LIN {X 0,Y 591.469,Z 583.737,A -85,B 0,C 180,E1 -8891.352,E2 -8891.352} C_VEL
LIN {X 0,Y 591.483,Z 583.74,A -85,B 0,C 180,E1 -8894.195,E2 -8894.195} C_VEL
LIN {X 0,Y 591.491,Z 583.733,A -85,B 0,C 180,E1 -8896.997,E2 -8896.997} C_VEL
LIN {X 0,Y 591.518,Z 583.737,A -85,B 0,C 180,E1 -8899.769,E2 -8899.769} C_VEL
LIN {X 0,Y 591.543,Z 583.729,A -85,B 0,C 180,E1 -8902.516,E2 -8902.516} C_VEL
LIN {X 0,Y 591.625,Z 583.717,A -85,B 0,C 180,E1 -8905.246,E2 -8905.246} C_VEL
LIN {X 0,Y 591.718,Z 583.706,A -85,B 0,C 180,E1 -8909.322,E2 -8909.322} C_VEL
LIN {X 0,Y 591.68,Z 583.711,A -85,B 0,C 180,E1 -8911.357,E2 -8911.357} C_VEL
LIN {X 0,Y 591.625,Z 583.717,A -85,B 0,C 180,E1 -8914.754,E2 -8914.754} C_VEL
LIN {X 0,Y 591.543,Z 583.729,A -85,B 0,C 180,E1 -8917.484,E2 -8917.484} C_VEL
LIN {X 0,Y 591.53,Z 583.729,A -85,B 0,C 180,E1 -8920.638,E2 -8920.638} C_VEL
LIN {X 0,Y 591.518,Z 583.738,A -85,B 0,C 180,E1 -8923.834,E2 -8923.834} C_VEL
LIN {X 0,Y 591.492,Z 583.735,A -85,B 0,C 180,E1 -8926.511,E2 -8926.511} C_VEL
LIN {X 0,Y 591.458,Z 583.739,A -85,B 0,C 180,E1 -8929.365,E2 -8929.365} C_VEL
LIN {X 0,Y 591.478,Z 583.738,A -85,B 0,C 180,E1 -8931.537,E2 -8931.537} C_VEL
LIN {X 0,Y 591.433,Z 583.743,A -85,B 0,C 180,E1 -8934.488,E2 -8934.488} C_VEL
LIN {X 0,Y 591.429,Z 583.744,A -85,B 0,C 180,E1 -8937.509,E2 -8937.509} C_VEL
LIN {X 0,Y 591.468,Z 583.742,A -85,B 0,C 180,E1 -8940.175,E2 -8940.175} C_VEL
LIN {X 0,Y 591.437,Z 583.74,A -85,B 0,C 180,E1 -8943.01,E2 -8943.01} C_VEL
LIN {X 0,Y 591.485,Z 583.737,A -85,B 0,C 180,E1 -8945.469,E2 -8945.469} C_VEL
LIN {X 0,Y 591.444,Z 583.749,A -85,B 0,C 180,E1 -8948.012,E2 -8948.012} C_VEL
LIN {X 0,Y 591.448,Z 583.739,A -85,B 0,C 180,E1 -8950.717,E2 -8950.717} C_VEL
LIN {X 0,Y 591.417,Z 583.744,A -85,B 0,C 180,E1 -8953.387,E2 -8953.387} C_VEL
LIN {X 0,Y 591.427,Z 583.746,A -85,B 0,C 180,E1 -8956.256,E2 -8956.256} C_VEL
LIN {X 0,Y 591.433,Z 583.743,A -85,B 0,C 180,E1 -8958.455,E2 -8958.455} C_VEL
LIN {X 0,Y 591.427,Z 583.743,A -85,B 0,C 180,E1 -8961.412,E2 -8961.412} C_VEL
LIN {X 0,Y 591.476,Z 583.741,A -85,B 0,C 180,E1 -8963.693,E2 -8963.693} C_VEL
LIN {X 0,Y 591.442,Z 583.746,A -85,B 0,C 180,E1 -8966.178,E2 -8966.178} C_VEL
LIN {X 0,Y 591.449,Z 583.74,A -85,B 0,C 180,E1 -8968.595,E2 -8968.595} C_VEL
LIN {X 0,Y 591.486,Z 583.734,A -85,B 0,C 180,E1 -8971.201,E2 -8971.201} C_VEL
LIN {X 0,Y 591.406,Z 583.75,A -85,B 0,C 180,E1 -8974.174,E2 -8974.174} C_VEL
LIN {X 0,Y 591.446,Z 583.744,A -85,B 0,C 180,E1 -8976.256,E2 -8976.256} C_VEL
LIN {X 0,Y 591.471,Z 583.738,A -85,B 0,C 180,E1 -8978.463,E2 -8978.463} C_VEL
LIN {X 0,Y 591.445,Z 583.741,A -85,B 0,C 180,E1 -8981.352,E2 -8981.352} C_VEL
LIN {X 0,Y 591.468,Z 583.742,A -85,B 0,C 180,E1 -8984.195,E2 -8984.195} C_VEL
LIN {X 0,Y 591.506,Z 583.736,A -85,B 0,C 180,E1 -8986.301,E2 -8986.301} C_VEL
LIN {X 0,Y 591.537,Z 583.729,A -85,B 0,C 180,E1 -8989.361,E2 -8989.361} C_VEL
LIN {X 0,Y 591.547,Z 583.728,A -85,B 0,C 180,E1 -8992.516,E2 -8992.516} C_VEL
LIN {X 0,Y 591.544,Z 583.728,A -85,B 0,C 180,E1 -8994.565,E2 -8994.565} C_VEL
LIN {X 0,Y 591.613,Z 583.728,A -85,B 0,C 180,E1 -8995.927,E2 -8995.927} C_VEL
LIN {X 0,Y 591.704,Z 583.708,A -85,B 0,C 180,E1 -8999.322,E2 -8999.322} C_VEL
LIN {X 0,Y 591.669,Z 583.713,A -85,B 0,C 180,E1 -9001.357,E2 -9001.357} C_VEL
LIN {X 0,Y 591.611,Z 583.718,A -85,B 0,C 180,E1 -9004.754,E2 -9004.754} C_VEL
LIN {X 0,Y 591.567,Z 583.724,A -85,B 0,C 180,E1 -9006.8,E2 -9006.8} C_VEL
LIN {X 0,Y 591.504,Z 583.735,A -85,B 0,C 180,E1 -9009.543,E2 -9009.543} C_VEL
LIN {X 0,Y 591.462,Z 583.741,A -85,B 0,C 180,E1 -9011.615,E2 -9011.615} C_VEL
LIN {X 0,Y 591.463,Z 583.74,A -85,B 0,C 180,E1 -9014.4,E2 -9014.4} C_VEL
LIN {X 0,Y 591.43,Z 583.741,A -85,B 0,C 180,E1 -9017.222,E2 -9017.222} C_VEL
LIN {X 0,Y 591.415,Z 583.744,A -85,B 0,C 180,E1 -9019.367,E2 -9019.367} C_VEL
LIN {X 0,Y 591.468,Z 583.741,A -85,B 0,C 180,E1 -9022.269,E2 -9022.269} C_VEL
LIN {X 0,Y 591.407,Z 583.745,A -85,B 0,C 180,E1 -9025.238,E2 -9025.238} C_VEL
LIN {X 0,Y 591.43,Z 583.744,A -85,B 0,C 180,E1 -9027.509,E2 -9027.509} C_VEL
LIN {X 0,Y 591.408,Z 583.752,A -85,B 0,C 180,E1 -9029.83,E2 -9029.83} C_VEL
LIN {X 0,Y 591.407,Z 583.749,A -85,B 0,C 180,E1 -9032.206,E2 -9032.206} C_VEL
LIN {X 0,Y 591.397,Z 583.746,A -85,B 0,C 180,E1 -9034.646,E2 -9034.646} C_VEL
LIN {X 0,Y 591.405,Z 583.744,A -85,B 0,C 180,E1 -9037.159,E2 -9037.159} C_VEL
LIN {X 0,Y 591.404,Z 583.751,A -85,B 0,C 180,E1 -9039.759,E2 -9039.759} C_VEL
LIN {X 0,Y 591.416,Z 583.743,A -85,B 0,C 180,E1 -9042.752,E2 -9042.752} C_VEL
LIN {X 0,Y 591.427,Z 583.747,A -85,B 0,C 180,E1 -9045.673,E2 -9045.673} C_VEL
LIN {X 0,Y 591.392,Z 583.748,A -85,B 0,C 180,E1 -9048.451,E2 -9048.451} C_VEL
LIN {X 0,Y 591.405,Z 583.744,A -85,B 0,C 180,E1 -9051.118,E2 -9051.118} C_VEL
LIN {X 0,Y 591.446,Z 583.745,A -85,B 0,C 180,E1 -9053.691,E2 -9053.691} C_VEL
LIN {X 0,Y 591.423,Z 583.748,A -85,B 0,C 180,E1 -9056.176,E2 -9056.176} C_VEL
LIN {X 0,Y 591.418,Z 583.743,A -85,B 0,C 180,E1 -9058.593,E2 -9058.593} C_VEL
LIN {X 0,Y 591.436,Z 583.741,A -85,B 0,C 180,E1 -9061.21,E2 -9061.21} C_VEL
LIN {X 0,Y 591.401,Z 583.755,A -85,B 0,C 180,E1 -9064.01,E2 -9064.01} C_VEL
LIN {X 0,Y 591.454,Z 583.794,A -85,B 0,C 180,E1 -9066.765,E2 -9066.765} C_VEL
LIN {X 0,Y 593.313,Z 594.595,A -85,B 0,C 180,E1 -9068.533,E2 -9068.533} C_VEL
LIN {X 0,Y 592.679,Z 611.185,A -85,B 0,C 180,E1 -9071.09,E2 -9071.09} C_VEL
LIN {X 0,Y 591.965,Z 630.482,A -85,B 0,C 180,E1 -9074.032,E2 -9074.032} C_VEL
LIN {X 0,Y 591.494,Z 647.827,A -85,B 0,C 180,E1 -9076.649,E2 -9076.649} C_VEL
LIN {X 0,Y 593.595,Z 665.618,A -85,B 0,C 180,E1 -9076.936,E2 -9076.936} C_VEL
LIN {X 0,Y 592.889,Z 754.339,A -85,B 0,C 180,E1 -9078.112,E2 -9078.112} C_VEL
LIN {X 0,Y 592.757,Z 763.761,A -85,B 0,C 180,E1 -9078.303,E2 -9078.303} C_VEL
LIN {X 0,Y 592.554,Z 773.554,A -85,B 0,C 180,E1 -9078.58,E2 -9078.58} C_VEL
LIN {X 0,Y 592.29,Z 784.736,A -85,B 0,C 180,E1 -9079.007,E2 -9079.007} C_VEL
LIN {X 0,Y 592.068,Z 795.202,A -85,B 0,C 180,E1 -9079.52,E2 -9079.52} C_VEL
LIN {X 0,Y 591.759,Z 803.814,A -85,B 0,C 180,E1 -9080.031,E2 -9080.031} C_VEL
LIN {X 0,Y 591.445,Z 813.28,A -85,B 0,C 180,E1 -9080.714,E2 -9080.714} C_VEL
LIN {X 0,Y 591.111,Z 822.077,A -85,B 0,C 180,E1 -9081.482,E2 -9081.482} C_VEL
LIN {X 0,Y 590.911,Z 828.739,A -85,B 0,C 180,E1 -9082.165,E2 -9082.165} C_VEL
LIN {X 0,Y 590.718,Z 835.721,A -85,B 0,C 180,E1 -9083.019,E2 -9083.019} C_VEL
LIN {X 0,Y 590.534,Z 841.558,A -85,B 0,C 180,E1 -9083.872,E2 -9083.872} C_VEL
LIN {X 0,Y 590.421,Z 847.209,A -85,B 0,C 180,E1 -9084.895,E2 -9084.895} C_VEL
LIN {X 0,Y 590.361,Z 851.655,A -85,B 0,C 180,E1 -9085.918,E2 -9085.918} C_VEL
LIN {X 0,Y 590.354,Z 853.992,A -85,B 0,C 180,E1 -9086.599,E2 -9086.599} C_VEL
LIN {X 0,Y 590.25,Z 857.375,A -85,B 0,C 180,E1 -9087.96,E2 -9087.96} C_VEL
LIN {X 0,Y 590.293,Z 858.953,A -85,B 0,C 180,E1 -9089.32,E2 -9089.32} C_VEL
LIN {X 0,Y 590.279,Z 859.252,A -85,B 0,C 180,E1 -9090,E2 -9090} C_VEL
LIN {X 0,Y 590.251,Z 858.372,A -85,B 0,C 180,E1 -9091.36,E2 -9091.36} C_VEL
LIN {X 0,Y 590.25,Z 857.378,A -85,B 0,C 180,E1 -9092.04,E2 -9092.04} C_VEL
LIN {X 0,Y 590.355,Z 854.043,A -85,B 0,C 180,E1 -9093.401,E2 -9093.401} C_VEL
LIN {X 0,Y 590.346,Z 850.416,A -85,B 0,C 180,E1 -9094.409,E2 -9094.409} C_VEL
LIN {X 0,Y 590.497,Z 845.517,A -85,B 0,C 180,E1 -9095.445,E2 -9095.445} C_VEL
LIN {X 0,Y 590.616,Z 839.39,A -85,B 0,C 180,E1 -9096.469,E2 -9096.469} C_VEL
LIN {X 0,Y 590.772,Z 833.183,A -85,B 0,C 180,E1 -9097.323,E2 -9097.323} C_VEL
LIN {X 0,Y 591.009,Z 825.7,A -85,B 0,C 180,E1 -9098.176,E2 -9098.176} C_VEL
LIN {X 0,Y 591.313,Z 816.604,A -85,B 0,C 180,E1 -9099.03,E2 -9099.03} C_VEL
LIN {X 0,Y 591.633,Z 807.844,A -85,B 0,C 180,E1 -9099.713,E2 -9099.713} C_VEL
LIN {X 0,Y 592.005,Z 798.651,A -85,B 0,C 180,E1 -9100.309,E2 -9100.309} C_VEL
LIN {X 0,Y 592.233,Z 788.554,A -85,B 0,C 180,E1 -9100.847,E2 -9100.847} C_VEL
LIN {X 0,Y 592.426,Z 779.278,A -85,B 0,C 180,E1 -9101.249,E2 -9101.249} C_VEL
LIN {X 0,Y 592.652,Z 767.637,A -85,B 0,C 180,E1 -9101.634,E2 -9101.634} C_VEL
LIN {X 0,Y 592.965,Z 756.804,A -85,B 0,C 180,E1 -9101.887,E2 -9101.887} C_VEL
LIN {X 0,Y 593.133,Z 737.904,A -85,B 0,C 180,E1 -9102.165,E2 -9102.165} C_VEL
LIN {X 0,Y 593.732,Z 664.622,A -85,B 0,C 180,E1 -9103.148,E2 -9103.148} C_VEL
LIN {X 0,Y 591.478,Z 647.186,A -85,B 0,C 180,E1 -9103.461,E2 -9103.461} C_VEL
LIN {X 0,Y 592.031,Z 629.576,A -85,B 0,C 180,E1 -9106.143,E2 -9106.143} C_VEL
LIN {X 0,Y 592.785,Z 610.85,A -85,B 0,C 180,E1 -9109.04,E2 -9109.04} C_VEL
LIN {X 0,Y 593.446,Z 595.538,A -85,B 0,C 180,E1 -9111.463,E2 -9111.463} C_VEL
LIN {X 0,Y 592.277,Z 588.19,A -85,B 0,C 180,E1 -9112.713,E2 -9112.713} C_VEL
LIN {X 0,Y 591.429,Z 583.752,A -85,B 0,C 180,E1 -9113.514,E2 -9113.514} C_VEL
LIN {X 0,Y 591.402,Z 583.756,A -85,B 0,C 180,E1 -9115.991,E2 -9115.991} C_VEL
LIN {X 0,Y 591.437,Z 583.747,A -85,B 0,C 180,E1 -9118.79,E2 -9118.79} C_VEL
LIN {X 0,Y 591.415,Z 583.752,A -85,B 0,C 180,E1 -9121.49,E2 -9121.49} C_VEL
LIN {X 0,Y 591.41,Z 583.749,A -85,B 0,C 180,E1 -9123.998,E2 -9123.998} C_VEL
LIN {X 0,Y 591.488,Z 583.734,A -85,B 0,C 180,E1 -9126.365,E2 -9126.365} C_VEL
LIN {X 0,Y 591.407,Z 583.743,A -85,B 0,C 180,E1 -9128.882,E2 -9128.882} C_VEL
LIN {X 0,Y 591.426,Z 583.746,A -85,B 0,C 180,E1 -9131.744,E2 -9131.744} C_VEL
LIN {X 0,Y 591.425,Z 583.745,A -85,B 0,C 180,E1 -9134.716,E2 -9134.716} C_VEL
LIN {X 0,Y 591.446,Z 583.746,A -85,B 0,C 180,E1 -9137.542,E2 -9137.542} C_VEL
LIN {X 0,Y 591.424,Z 583.744,A -85,B 0,C 180,E1 -9140.338,E2 -9140.338} C_VEL
LIN {X 0,Y 591.452,Z 583.745,A -85,B 0,C 180,E1 -9142.844,E2 -9142.844} C_VEL
LIN {X 0,Y 591.454,Z 583.744,A -85,B 0,C 180,E1 -9145.358,E2 -9145.358} C_VEL
LIN {X 0,Y 591.44,Z 583.741,A -85,B 0,C 180,E1 -9147.796,E2 -9147.796} C_VEL
LIN {X 0,Y 591.447,Z 583.741,A -85,B 0,C 180,E1 -9150.172,E2 -9150.172} C_VEL
LIN {X 0,Y 591.433,Z 583.75,A -85,B 0,C 180,E1 -9152.653,E2 -9152.653} C_VEL
LIN {X 0,Y 591.461,Z 583.74,A -85,B 0,C 180,E1 -9155.767,E2 -9155.767} C_VEL
LIN {X 0,Y 591.475,Z 583.746,A -85,B 0,C 180,E1 -9158.462,E2 -9158.462} C_VEL
LIN {X 0,Y 591.456,Z 583.744,A -85,B 0,C 180,E1 -9161.352,E2 -9161.352} C_VEL
LIN {X 0,Y 591.472,Z 583.746,A -85,B 0,C 180,E1 -9164.194,E2 -9164.194} C_VEL
LIN {X 0,Y 591.511,Z 583.741,A -85,B 0,C 180,E1 -9166.3,E2 -9166.3} C_VEL
LIN {X 0,Y 591.542,Z 583.828,A -85,B 0,C 180,E1 -9169.323,E2 -9169.323} C_VEL
LIN {X 0,Y 592.762,Z 591.438,A -85,B 0,C 180,E1 -9170.821,E2 -9170.821} C_VEL
LIN {X 0,Y 592.685,Z 598.772,A -85,B 0,C 180,E1 -9172.189,E2 -9172.189} C_VEL
LIN {X 0,Y 591.984,Z 615.621,A -85,B 0,C 180,E1 -9175.249,E2 -9175.249} C_VEL
LIN {X 0,Y 591.49,Z 623.222,A -85,B 0,C 180,E1 -9176.605,E2 -9176.605} C_VEL
LIN {X 0,Y 593.96,Z 637.425,A -85,B 0,C 180,E1 -9176.873,E2 -9176.873} C_VEL
LIN {X 0,Y 592.848,Z 729.098,A -85,B 0,C 180,E1 -9178.117,E2 -9178.117} C_VEL
LIN {X 0,Y 592.71,Z 738.945,A -85,B 0,C 180,E1 -9178.328,E2 -9178.328} C_VEL
LIN {X 0,Y 592.558,Z 748.292,A -85,B 0,C 180,E1 -9178.603,E2 -9178.603} C_VEL
LIN {X 0,Y 592.408,Z 758.227,A -85,B 0,C 180,E1 -9178.984,E2 -9178.984} C_VEL
LIN {X 0,Y 592.266,Z 768.619,A -85,B 0,C 180,E1 -9179.492,E2 -9179.492} C_VEL
LIN {X 0,Y 591.96,Z 778.45,A -85,B 0,C 180,E1 -9180.085,E2 -9180.085} C_VEL
LIN {X 0,Y 591.672,Z 787.684,A -85,B 0,C 180,E1 -9180.763,E2 -9180.763} C_VEL
LIN {X 0,Y 591.351,Z 794.626,A -85,B 0,C 180,E1 -9181.357,E2 -9181.357} C_VEL
LIN {X 0,Y 591.05,Z 802.856,A -85,B 0,C 180,E1 -9182.207,E2 -9182.207} C_VEL
LIN {X 0,Y 590.823,Z 809.72,A -85,B 0,C 180,E1 -9183.058,E2 -9183.058} C_VEL
LIN {X 0,Y 590.596,Z 814.438,A -85,B 0,C 180,E1 -9183.74,E2 -9183.74} C_VEL
LIN {X 0,Y 590.517,Z 820.801,A -85,B 0,C 180,E1 -9184.881,E2 -9184.881} C_VEL
LIN {X 0,Y 590.415,Z 825.031,A -85,B 0,C 180,E1 -9185.849,E2 -9185.849} C_VEL
LIN {X 0,Y 590.334,Z 828.296,A -85,B 0,C 180,E1 -9186.814,E2 -9186.814} C_VEL
LIN {X 0,Y 590.208,Z 831.28,A -85,B 0,C 180,E1 -9188.187,E2 -9188.187} C_VEL
LIN {X 0,Y 590.224,Z 832.247,A -85,B 0,C 180,E1 -9188.875,E2 -9188.875} C_VEL
LIN {X 0,Y 590.249,Z 832.726,A -85,B 0,C 180,E1 -9190.253,E2 -9190.253} C_VEL
LIN {X 0,Y 590.208,Z 832.384,A -85,B 0,C 180,E1 -9190.946,E2 -9190.946} C_VEL
LIN {X 0,Y 590.232,Z 830.382,A -85,B 0,C 180,E1 -9192.334,E2 -9192.334} C_VEL
LIN {X 0,Y 590.338,Z 827.785,A -85,B 0,C 180,E1 -9193.358,E2 -9193.358} C_VEL
LIN {X 0,Y 590.392,Z 823.957,A -85,B 0,C 180,E1 -9194.427,E2 -9194.427} C_VEL
LIN {X 0,Y 590.559,Z 818.983,A -85,B 0,C 180,E1 -9195.478,E2 -9195.478} C_VEL
LIN {X 0,Y 590.675,Z 814.487,A -85,B 0,C 180,E1 -9196.262,E2 -9196.262} C_VEL
LIN {X 0,Y 590.838,Z 807.579,A -85,B 0,C 180,E1 -9197.24,E2 -9197.24} C_VEL
LIN {X 0,Y 591.136,Z 799.984,A -85,B 0,C 180,E1 -9198.12,E2 -9198.12} C_VEL
LIN {X 0,Y 591.418,Z 790.622,A -85,B 0,C 180,E1 -9199.007,E2 -9199.007} C_VEL
LIN {X 0,Y 591.632,Z 782.823,A -85,B 0,C 180,E1 -9199.629,E2 -9199.629} C_VEL
LIN {X 0,Y 591.952,Z 773.479,A -85,B 0,C 180,E1 -9200.249,E2 -9200.249} C_VEL
LIN {X 0,Y 592.282,Z 762.523,A -85,B 0,C 180,E1 -9200.836,E2 -9200.836} C_VEL
LIN {X 0,Y 592.465,Z 753.324,A -85,B 0,C 180,E1 -9201.235,E2 -9201.235} C_VEL
LIN {X 0,Y 592.606,Z 742.156,A -85,B 0,C 180,E1 -9201.608,E2 -9201.608} C_VEL
LIN {X 0,Y 592.878,Z 731.012,A -85,B 0,C 180,E1 -9201.871,E2 -9201.871} C_VEL
LIN {X 0,Y 593.071,Z 712.766,A -85,B 0,C 180,E1 -9202.137,E2 -9202.137} C_VEL
LIN {X 0,Y 593.631,Z 636.363,A -85,B 0,C 180,E1 -9203.142,E2 -9203.142} C_VEL
LIN {X 0,Y 591.498,Z 622.471,A -85,B 0,C 180,E1 -9203.375,E2 -9203.375} C_VEL
LIN {X 0,Y 591.983,Z 605.586,A -85,B 0,C 180,E1 -9206.34,E2 -9206.34} C_VEL
LIN {X 0,Y 592.455,Z 590.653,A -85,B 0,C 180,E1 -9208.994,E2 -9208.994} C_VEL
LIN {X 0,Y 591.515,Z 583.74,A -85,B 0,C 180,E1 -9210.305,E2 -9210.305} C_VEL
LIN {X 0,Y 591.428,Z 583.741,A -85,B 0,C 180,E1 -9213.01,E2 -9213.01} C_VEL
LIN {X 0,Y 591.467,Z 583.739,A -85,B 0,C 180,E1 -9215.47,E2 -9215.47} C_VEL
LIN {X 0,Y 591.418,Z 583.752,A -85,B 0,C 180,E1 -9218.014,E2 -9218.014} C_VEL
LIN {X 0,Y 591.45,Z 583.739,A -85,B 0,C 180,E1 -9220.717,E2 -9220.717} C_VEL
LIN {X 0,Y 591.419,Z 583.744,A -85,B 0,C 180,E1 -9223.386,E2 -9223.386} C_VEL
LIN {X 0,Y 591.429,Z 583.746,A -85,B 0,C 180,E1 -9226.255,E2 -9226.255} C_VEL
LIN {X 0,Y 591.434,Z 583.743,A -85,B 0,C 180,E1 -9228.454,E2 -9228.454} C_VEL
LIN {X 0,Y 591.409,Z 583.743,A -85,B 0,C 180,E1 -9231.118,E2 -9231.118} C_VEL
LIN {X 0,Y 591.476,Z 583.74,A -85,B 0,C 180,E1 -9233.692,E2 -9233.692} C_VEL
LIN {X 0,Y 591.441,Z 583.746,A -85,B 0,C 180,E1 -9236.177,E2 -9236.177} C_VEL
LIN {X 0,Y 591.428,Z 583.746,A -85,B 0,C 180,E1 -9237.98,E2 -9237.98} C_VEL
LIN {X 0,Y 590.757,Z 583.827,A -85,B 0,C 180,E1 -9238.549,E2 -9238.549} C_VEL
LIN {X 0,Y 587.894,Z 584.184,A -85,B 0,C 180,E1 -9239.471,E2 -9239.471} C_VEL
LIN {X 0,Y 585.493,Z 584.486,A -85,B 0,C 180,E1 -9240.213,E2 -9240.213} C_VEL
LIN {X 0,Y 584.485,Z 584.606,A -85,B 0,C 180,E1 -9240.786,E2 -9240.786} C_VEL
LIN {X 0,Y 584.415,Z 584.614,A -85,B 0,C 180,E1 -9240.98,E2 -9240.98} C_VEL
LIN {X 0,Y 584.385,Z 584.624,A -85,B 0,C 180,E1 -9243.674,E2 -9243.674} C_VEL
LIN {X 0,Y 584.427,Z 584.623,A -85,B 0,C 180,E1 -9245.952,E2 -9245.952} C_VEL
LIN {X 0,Y 584.442,Z 584.611,A -85,B 0,C 180,E1 -9248.928,E2 -9248.928} C_VEL
LIN {X 0,Y 584.405,Z 584.624,A -85,B 0,C 180,E1 -9251.843,E2 -9251.843} C_VEL
LIN {X 0,Y 584.429,Z 584.623,A -85,B 0,C 180,E1 -9253.999,E2 -9253.999} C_VEL
LIN {X 0,Y 584.468,Z 584.608,A -85,B 0,C 180,E1 -9256.838,E2 -9256.838} C_VEL
LIN {X 0,Y 584.474,Z 584.612,A -85,B 0,C 180,E1 -9259.644,E2 -9259.644} C_VEL
LIN {X 0,Y 584.519,Z 584.604,A -85,B 0,C 180,E1 -9262.425,E2 -9262.425} C_VEL
LIN {X 0,Y 584.596,Z 584.592,A -85,B 0,C 180,E1 -9265.189,E2 -9265.189} C_VEL
LIN {X 0,Y 584.692,Z 584.581,A -85,B 0,C 180,E1 -9269.313,E2 -9269.313} C_VEL
LIN {X 0,Y 584.627,Z 584.59,A -85,B 0,C 180,E1 -9271.373,E2 -9271.373} C_VEL
LIN {X 0,Y 584.596,Z 584.592,A -85,B 0,C 180,E1 -9274.811,E2 -9274.811} C_VEL
LIN {X 0,Y 584.519,Z 584.606,A -85,B 0,C 180,E1 -9277.574,E2 -9277.574} C_VEL
LIN {X 0,Y 584.491,Z 584.606,A -85,B 0,C 180,E1 -9280.684,E2 -9280.684} C_VEL
LIN {X 0,Y 584.478,Z 584.616,A -85,B 0,C 180,E1 -9283.903,E2 -9283.903} C_VEL
LIN {X 0,Y 584.448,Z 584.611,A -85,B 0,C 180,E1 -9286.716,E2 -9286.716} C_VEL
LIN {X 0,Y 584.41,Z 584.62,A -85,B 0,C 180,E1 -9289.609,E2 -9289.609} C_VEL
LIN {X 0,Y 584.446,Z 584.618,A -85,B 0,C 180,E1 -9291.81,E2 -9291.81} C_VEL
LIN {X 0,Y 584.387,Z 584.618,A -85,B 0,C 180,E1 -9294.803,E2 -9294.803} C_VEL
LIN {X 0,Y 584.397,Z 584.625,A -85,B 0,C 180,E1 -9297.868,E2 -9297.868} C_VEL
LIN {X 0,Y 584.414,Z 584.618,A -85,B 0,C 180,E1 -9300.352,E2 -9300.352} C_VEL
LIN {X 0,Y 584.399,Z 584.616,A -85,B 0,C 180,E1 -9302.966,E2 -9302.966} C_VEL
LIN {X 0,Y 584.421,Z 584.624,A -85,B 0,C 180,E1 -9305.964,E2 -9305.964} C_VEL
LIN {X 0,Y 584.381,Z 584.62,A -85,B 0,C 180,E1 -9308.556,E2 -9308.556} C_VEL
LIN {X 0,Y 584.379,Z 584.62,A -85,B 0,C 180,E1 -9311.242,E2 -9311.242} C_VEL
LIN {X 0,Y 584.391,Z 584.626,A -85,B 0,C 180,E1 -9314.042,E2 -9314.042} C_VEL
LIN {X 0,Y 584.394,Z 584.617,A -85,B 0,C 180,E1 -9316.982,E2 -9316.982} C_VEL
LIN {X 0,Y 584.409,Z 584.621,A -85,B 0,C 180,E1 -9319.668,E2 -9319.668} C_VEL
LIN {X 0,Y 584.43,Z 584.617,A -85,B 0,C 180,E1 -9322.321,E2 -9322.321} C_VEL
LIN {X 0,Y 584.419,Z 584.614,A -85,B 0,C 180,E1 -9324.88,E2 -9324.88} C_VEL
LIN {X 0,Y 584.385,Z 584.62,A -85,B 0,C 180,E1 -9327.36,E2 -9327.36} C_VEL
LIN {X 0,Y 584.423,Z 584.621,A -85,B 0,C 180,E1 -9329.777,E2 -9329.777} C_VEL
LIN {X 0,Y 584.396,Z 584.619,A -85,B 0,C 180,E1 -9332.492,E2 -9332.492} C_VEL
LIN {X 0,Y 584.413,Z 584.619,A -85,B 0,C 180,E1 -9335.629,E2 -9335.629} C_VEL
LIN {X 0,Y 584.442,Z 584.617,A -85,B 0,C 180,E1 -9338.19,E2 -9338.19} C_VEL
LIN {X 0,Y 584.409,Z 584.615,A -85,B 0,C 180,E1 -9341.119,E2 -9341.119} C_VEL
LIN {X 0,Y 584.412,Z 584.625,A -85,B 0,C 180,E1 -9343.999,E2 -9343.999} C_VEL
LIN {X 0,Y 584.483,Z 584.613,A -85,B 0,C 180,E1 -9346.133,E2 -9346.133} C_VEL
LIN {X 0,Y 584.501,Z 584.605,A -85,B 0,C 180,E1 -9349.313,E2 -9349.313} C_VEL
LIN {X 0,Y 584.523,Z 584.604,A -85,B 0,C 180,E1 -9352.426,E2 -9352.426} C_VEL
LIN {X 0,Y 584.505,Z 584.605,A -85,B 0,C 180,E1 -9354.499,E2 -9354.499} C_VEL
LIN {X 0,Y 584.578,Z 584.603,A -85,B 0,C 180,E1 -9355.878,E2 -9355.878} C_VEL
LIN {X 0,Y 584.68,Z 584.583,A -85,B 0,C 180,E1 -9359.314,E2 -9359.314} C_VEL
LIN {X 0,Y 584.617,Z 584.591,A -85,B 0,C 180,E1 -9361.373,E2 -9361.373} C_VEL
LIN {X 0,Y 584.582,Z 584.594,A -85,B 0,C 180,E1 -9364.811,E2 -9364.811} C_VEL
LIN {X 0,Y 584.531,Z 584.6,A -85,B 0,C 180,E1 -9366.882,E2 -9366.882} C_VEL
LIN {X 0,Y 584.483,Z 584.611,A -85,B 0,C 180,E1 -9369.659,E2 -9369.659} C_VEL
LIN {X 0,Y 584.437,Z 584.619,A -85,B 0,C 180,E1 -9371.756,E2 -9371.756} C_VEL
LIN {X 0,Y 584.43,Z 584.614,A -85,B 0,C 180,E1 -9374.577,E2 -9374.577} C_VEL
LIN {X 0,Y 584.383,Z 584.621,A -85,B 0,C 180,E1 -9377.437,E2 -9377.437} C_VEL
LIN {X 0,Y 584.401,Z 584.62,A -85,B 0,C 180,E1 -9380.34,E2 -9380.34} C_VEL
LIN {X 0,Y 584.413,Z 584.616,A -85,B 0,C 180,E1 -9382.65,E2 -9382.65} C_VEL
LIN {X 0,Y 584.384,Z 584.619,A -85,B 0,C 180,E1 -9384.804,E2 -9384.804} C_VEL
LIN {X 0,Y 584.396,Z 584.626,A -85,B 0,C 180,E1 -9387.869,E2 -9387.869} C_VEL
LIN {X 0,Y 584.355,Z 584.626,A -85,B 0,C 180,E1 -9390.341,E2 -9390.341} C_VEL
LIN {X 0,Y 584.365,Z 584.621,A -85,B 0,C 180,E1 -9392.96,E2 -9392.96} C_VEL
LIN {X 0,Y 584.385,Z 584.629,A -85,B 0,C 180,E1 -9395.967,E2 -9395.967} C_VEL
LIN {X 0,Y 584.359,Z 584.622,A -85,B 0,C 180,E1 -9398.82,E2 -9398.82} C_VEL
LIN {X 0,Y 584.342,Z 584.625,A -85,B 0,C 180,E1 -9401.245,E2 -9401.245} C_VEL
LIN {X 0,Y 584.392,Z 584.626,A -85,B 0,C 180,E1 -9404.042,E2 -9404.042} C_VEL
LIN {X 0,Y 584.389,Z 584.618,A -85,B 0,C 180,E1 -9406.982,E2 -9406.982} C_VEL
LIN {X 0,Y 584.355,Z 584.63,A -85,B 0,C 180,E1 -9410.098,E2 -9410.098} C_VEL
LIN {X 0,Y 584.37,Z 584.624,A -85,B 0,C 180,E1 -9412.316,E2 -9412.316} C_VEL
LIN {X 0,Y 584.371,Z 584.62,A -85,B 0,C 180,E1 -9414.877,E2 -9414.877} C_VEL
LIN {X 0,Y 584.353,Z 584.624,A -85,B 0,C 180,E1 -9417.357,E2 -9417.357} C_VEL
LIN {X 0,Y 584.365,Z 584.628,A -85,B 0,C 180,E1 -9419.773,E2 -9419.773} C_VEL
LIN {X 0,Y 584.387,Z 584.62,A -85,B 0,C 180,E1 -9422.494,E2 -9422.494} C_VEL
LIN {X 0,Y 584.394,Z 584.627,A -85,B 0,C 180,E1 -9425.633,E2 -9425.633} C_VEL
LIN {X 0,Y 584.415,Z 584.736,A -85,B 0,C 180,E1 -9426.655,E2 -9426.655} C_VEL
LIN {X 0,Y 586.191,Z 594.368,A -85,B 0,C 180,E1 -9428.259,E2 -9428.259} C_VEL
LIN {X 0,Y 586.089,Z 601.33,A -85,B 0,C 180,E1 -9429.356,E2 -9429.356} C_VEL
LIN {X 0,Y 585.416,Z 617.535,A -85,B 0,C 180,E1 -9431.875,E2 -9431.875} C_VEL
LIN {X 0,Y 584.708,Z 638.366,A -85,B 0,C 180,E1 -9435.075,E2 -9435.075} C_VEL
LIN {X 0,Y 584.459,Z 647.971,A -85,B 0,C 180,E1 -9436.507,E2 -9436.507} C_VEL
LIN {X 0,Y 586.658,Z 666.038,A -85,B 0,C 180,E1 -9436.8,E2 -9436.8} C_VEL
LIN {X 0,Y 585.912,Z 754.072,A -85,B 0,C 180,E1 -9437.99,E2 -9437.99} C_VEL
LIN {X 0,Y 585.726,Z 764.324,A -85,B 0,C 180,E1 -9438.205,E2 -9438.205} C_VEL
LIN {X 0,Y 585.546,Z 773.92,A -85,B 0,C 180,E1 -9438.486,E2 -9438.486} C_VEL
LIN {X 0,Y 585.286,Z 784.05,A -85,B 0,C 180,E1 -9438.874,E2 -9438.874} C_VEL
LIN {X 0,Y 585.055,Z 794.914,A -85,B 0,C 180,E1 -9439.41,E2 -9439.41} C_VEL
LIN {X 0,Y 584.703,Z 804.541,A -85,B 0,C 180,E1 -9439.997,E2 -9439.997} C_VEL
LIN {X 0,Y 584.416,Z 812.833,A -85,B 0,C 180,E1 -9440.602,E2 -9440.602} C_VEL
LIN {X 0,Y 584.082,Z 821.685,A -85,B 0,C 180,E1 -9441.379,E2 -9441.379} C_VEL
LIN {X 0,Y 583.803,Z 829.826,A -85,B 0,C 180,E1 -9442.243,E2 -9442.243} C_VEL
LIN {X 0,Y 583.603,Z 836.6,A -85,B 0,C 180,E1 -9443.107,E2 -9443.107} C_VEL
LIN {X 0,Y 583.46,Z 841.28,A -85,B 0,C 180,E1 -9443.797,E2 -9443.797} C_VEL
LIN {X 0,Y 583.342,Z 846.966,A -85,B 0,C 180,E1 -9444.833,E2 -9444.833} C_VEL
LIN {X 0,Y 583.267,Z 851.437,A -85,B 0,C 180,E1 -9445.868,E2 -9445.868} C_VEL
LIN {X 0,Y 583.268,Z 853.776,A -85,B 0,C 180,E1 -9446.558,E2 -9446.558} C_VEL
LIN {X 0,Y 583.161,Z 857.193,A -85,B 0,C 180,E1 -9447.935,E2 -9447.935} C_VEL
LIN {X 0,Y 583.194,Z 858.787,A -85,B 0,C 180,E1 -9449.312,E2 -9449.312} C_VEL
LIN {X 0,Y 583.182,Z 859.09,A -85,B 0,C 180,E1 -9450,E2 -9450} C_VEL
LIN {X 0,Y 583.153,Z 858.225,A -85,B 0,C 180,E1 -9451.377,E2 -9451.377} C_VEL
LIN {X 0,Y 583.162,Z 857.228,A -85,B 0,C 180,E1 -9452.065,E2 -9452.065} C_VEL
LIN {X 0,Y 583.268,Z 853.903,A -85,B 0,C 180,E1 -9453.443,E2 -9453.443} C_VEL
LIN {X 0,Y 583.25,Z 850.882,A -85,B 0,C 180,E1 -9454.318,E2 -9454.318} C_VEL
LIN {X 0,Y 583.421,Z 845.373,A -85,B 0,C 180,E1 -9455.512,E2 -9455.512} C_VEL
LIN {X 0,Y 583.533,Z 839.239,A -85,B 0,C 180,E1 -9456.548,E2 -9456.548} C_VEL
LIN {X 0,Y 583.718,Z 833.036,A -85,B 0,C 180,E1 -9457.412,E2 -9457.412} C_VEL
LIN {X 0,Y 583.952,Z 825.559,A -85,B 0,C 180,E1 -9458.276,E2 -9458.276} C_VEL
LIN {X 0,Y 584.295,Z 816.474,A -85,B 0,C 180,E1 -9459.14,E2 -9459.14} C_VEL
LIN {X 0,Y 584.645,Z 807.73,A -85,B 0,C 180,E1 -9459.83,E2 -9459.83} C_VEL
LIN {X 0,Y 585.025,Z 798.684,A -85,B 0,C 180,E1 -9460.426,E2 -9460.426} C_VEL
LIN {X 0,Y 585.205,Z 790.161,A -85,B 0,C 180,E1 -9460.9,E2 -9460.9} C_VEL
LIN {X 0,Y 585.467,Z 779.216,A -85,B 0,C 180,E1 -9461.385,E2 -9461.385} C_VEL
LIN {X 0,Y 585.715,Z 767.627,A -85,B 0,C 180,E1 -9461.774,E2 -9461.774} C_VEL
LIN {X 0,Y 586.023,Z 756.911,A -85,B 0,C 180,E1 -9462.03,E2 -9462.03} C_VEL
LIN {X 0,Y 586.222,Z 736.743,A -85,B 0,C 180,E1 -9462.332,E2 -9462.332} C_VEL
LIN {X 0,Y 586.832,Z 665.026,A -85,B 0,C 180,E1 -9463.319,E2 -9463.319} C_VEL
LIN {X 0,Y 584.468,Z 647.235,A -85,B 0,C 180,E1 -9463.636,E2 -9463.636} C_VEL
LIN {X 0,Y 585.053,Z 629.579,A -85,B 0,C 180,E1 -9466.341,E2 -9466.341} C_VEL
LIN {X 0,Y 585.878,Z 610.752,A -85,B 0,C 180,E1 -9469.304,E2 -9469.304} C_VEL
LIN {X 0,Y 586.495,Z 597.301,A -85,B 0,C 180,E1 -9471.465,E2 -9471.465} C_VEL
LIN {X 0,Y 585.671,Z 591.263,A -85,B 0,C 180,E1 -9472.502,E2 -9472.502} C_VEL
LIN {X 0,Y 584.386,Z 584.628,A -85,B 0,C 180,E1 -9473.697,E2 -9473.697} C_VEL
LIN {X 0,Y 584.351,Z 584.634,A -85,B 0,C 180,E1 -9476.328,E2 -9476.328} C_VEL
LIN {X 0,Y 584.384,Z 584.627,A -85,B 0,C 180,E1 -9478.957,E2 -9478.957} C_VEL
LIN {X 0,Y 584.379,Z 584.628,A -85,B 0,C 180,E1 -9481.829,E2 -9481.829} C_VEL
LIN {X 0,Y 584.39,Z 584.621,A -85,B 0,C 180,E1 -9484.287,E2 -9484.287} C_VEL
LIN {X 0,Y 584.403,Z 584.617,A -85,B 0,C 180,E1 -9486.819,E2 -9486.819} C_VEL
LIN {X 0,Y 584.359,Z 584.623,A -85,B 0,C 180,E1 -9489.902,E2 -9489.902} C_VEL
LIN {X 0,Y 584.399,Z 584.617,A -85,B 0,C 180,E1 -9492.16,E2 -9492.16} C_VEL
LIN {X 0,Y 584.394,Z 584.624,A -85,B 0,C 180,E1 -9495.005,E2 -9495.005} C_VEL
LIN {X 0,Y 584.411,Z 584.618,A -85,B 0,C 180,E1 -9497.996,E2 -9497.996} C_VEL
LIN {X 0,Y 584.365,Z 584.625,A -85,B 0,C 180,E1 -9500.559,E2 -9500.559} C_VEL
LIN {X 0,Y 584.439,Z 584.618,A -85,B 0,C 180,E1 -9503.417,E2 -9503.417} C_VEL
LIN {X 0,Y 584.404,Z 584.618,A -85,B 0,C 180,E1 -9505.793,E2 -9505.793} C_VEL
LIN {X 0,Y 584.408,Z 584.619,A -85,B 0,C 180,E1 -9508.318,E2 -9508.318} C_VEL
LIN {X 0,Y 584.431,Z 584.617,A -85,B 0,C 180,E1 -9511.354,E2 -9511.354} C_VEL
LIN {X 0,Y 584.359,Z 584.63,A -85,B 0,C 180,E1 -9514.436,E2 -9514.436} C_VEL
LIN {X 0,Y 584.402,Z 584.627,A -85,B 0,C 180,E1 -9516.701,E2 -9516.701} C_VEL
LIN {X 0,Y 584.441,Z 584.618,A -85,B 0,C 180,E1 -9519.2,E2 -9519.2} C_VEL
LIN {X 0,Y 584.401,Z 584.625,A -85,B 0,C 180,E1 -9521.843,E2 -9521.843} C_VEL
LIN {X 0,Y 584.433,Z 584.621,A -85,B 0,C 180,E1 -9524.712,E2 -9524.712} C_VEL
LIN {X 0,Y 584.461,Z 584.617,A -85,B 0,C 180,E1 -9526.838,E2 -9526.838} C_VEL
LIN {X 0,Y 584.494,Z 584.76,A -85,B 0,C 180,E1 -9529.159,E2 -9529.159} C_VEL
LIN {X 0,Y 585.79,Z 592.504,A -85,B 0,C 180,E1 -9530.71,E2 -9530.71} C_VEL
LIN {X 0,Y 585.738,Z 599.831,A -85,B 0,C 180,E1 -9532.095,E2 -9532.095} C_VEL
LIN {X 0,Y 584.985,Z 616.638,A -85,B 0,C 180,E1 -9535.192,E2 -9535.192} C_VEL
LIN {X 0,Y 584.57,Z 623.648,A -85,B 0,C 180,E1 -9536.425,E2 -9536.425} C_VEL
LIN {X 0,Y 587.134,Z 638.528,A -85,B 0,C 180,E1 -9536.708,E2 -9536.708} C_VEL
LIN {X 0,Y 585.937,Z 729.146,A -85,B 0,C 180,E1 -9537.966,E2 -9537.966} C_VEL
LIN {X 0,Y 585.774,Z 738.993,A -85,B 0,C 180,E1 -9538.18,E2 -9538.18} C_VEL
LIN {X 0,Y 585.596,Z 749.503,A -85,B 0,C 180,E1 -9538.5,E2 -9538.5} C_VEL
LIN {X 0,Y 585.427,Z 759.19,A -85,B 0,C 180,E1 -9538.886,E2 -9538.886} C_VEL
LIN {X 0,Y 585.271,Z 769.431,A -85,B 0,C 180,E1 -9539.4,E2 -9539.4} C_VEL
LIN {X 0,Y 585.005,Z 777.928,A -85,B 0,C 180,E1 -9539.914,E2 -9539.914} C_VEL
LIN {X 0,Y 584.693,Z 787.285,A -85,B 0,C 180,E1 -9540.6,E2 -9540.6} C_VEL
LIN {X 0,Y 584.255,Z 796.03,A -85,B 0,C 180,E1 -9541.374,E2 -9541.374} C_VEL
LIN {X 0,Y 584.036,Z 802.64,A -85,B 0,C 180,E1 -9542.062,E2 -9542.062} C_VEL
LIN {X 0,Y 583.805,Z 809.574,A -85,B 0,C 180,E1 -9542.923,E2 -9542.923} C_VEL
LIN {X 0,Y 583.529,Z 815.393,A -85,B 0,C 180,E1 -9543.785,E2 -9543.785} C_VEL
LIN {X 0,Y 583.435,Z 821.009,A -85,B 0,C 180,E1 -9544.82,E2 -9544.82} C_VEL
LIN {X 0,Y 583.336,Z 825.44,A -85,B 0,C 180,E1 -9545.858,E2 -9545.858} C_VEL
LIN {X 0,Y 583.241,Z 828.795,A -85,B 0,C 180,E1 -9546.897,E2 -9546.897} C_VEL
LIN {X 0,Y 583.142,Z 830.439,A -85,B 0,C 180,E1 -9547.592,E2 -9547.592} C_VEL
LIN {X 0,Y 583.128,Z 832.535,A -85,B 0,C 180,E1 -9548.983,E2 -9548.983} C_VEL
LIN {X 0,Y 583.17,Z 832.972,A -85,B 0,C 180,E1 -9549.968,E2 -9549.968} C_VEL
LIN {X 0,Y 583.128,Z 832.458,A -85,B 0,C 180,E1 -9551.08,E2 -9551.08} C_VEL
LIN {X 0,Y 583.17,Z 830.198,A -85,B 0,C 180,E1 -9552.485,E2 -9552.485} C_VEL
LIN {X 0,Y 583.244,Z 827.861,A -85,B 0,C 180,E1 -9553.401,E2 -9553.401} C_VEL
LIN {X 0,Y 583.297,Z 824.966,A -85,B 0,C 180,E1 -9554.251,E2 -9554.251} C_VEL
LIN {X 0,Y 583.439,Z 820.258,A -85,B 0,C 180,E1 -9555.314,E2 -9555.314} C_VEL
LIN {X 0,Y 583.604,Z 813.862,A -85,B 0,C 180,E1 -9556.429,E2 -9556.429} C_VEL
LIN {X 0,Y 583.787,Z 806.465,A -85,B 0,C 180,E1 -9557.455,E2 -9557.455} C_VEL
LIN {X 0,Y 584.103,Z 798.918,A -85,B 0,C 180,E1 -9558.314,E2 -9558.314} C_VEL
LIN {X 0,Y 584.374,Z 791.072,A -85,B 0,C 180,E1 -9559.064,E2 -9559.064} C_VEL
LIN {X 0,Y 584.633,Z 782.043,A -85,B 0,C 180,E1 -9559.783,E2 -9559.783} C_VEL
LIN {X 0,Y 584.937,Z 772.482,A -85,B 0,C 180,E1 -9560.411,E2 -9560.411} C_VEL
LIN {X 0,Y 585.273,Z 762.901,A -85,B 0,C 180,E1 -9560.927,E2 -9560.927} C_VEL
LIN {X 0,Y 585.46,Z 753.122,A -85,B 0,C 180,E1 -9561.355,E2 -9561.355} C_VEL
LIN {X 0,Y 585.612,Z 742.392,A -85,B 0,C 180,E1 -9561.718,E2 -9561.718} C_VEL
LIN {X 0,Y 585.9,Z 731.332,A -85,B 0,C 180,E1 -9561.983,E2 -9561.983} C_VEL
LIN {X 0,Y 586.101,Z 713.193,A -85,B 0,C 180,E1 -9562.252,E2 -9562.252} C_VEL
LIN {X 0,Y 586.727,Z 637.384,A -85,B 0,C 180,E1 -9563.271,E2 -9563.271} C_VEL
LIN {X 0,Y 584.477,Z 622.536,A -85,B 0,C 180,E1 -9563.535,E2 -9563.535} C_VEL
LIN {X 0,Y 584.981,Z 605.908,A -85,B 0,C 180,E1 -9566.488,E2 -9566.488} C_VEL
LIN {X 0,Y 585.441,Z 592.655,A -85,B 0,C 180,E1 -9568.867,E2 -9568.867} C_VEL
LIN {X 0,Y 584.8,Z 586.539,A -85,B 0,C 180,E1 -9570.004,E2 -9570.004} C_VEL
LIN {X 0,Y 584.496,Z 584.613,A -85,B 0,C 180,E1 -9570.394,E2 -9570.394} C_VEL
LIN {X 0,Y 584.382,Z 584.621,A -85,B 0,C 180,E1 -9573.46,E2 -9573.46} C_VEL
LIN {X 0,Y 584.418,Z 584.625,A -85,B 0,C 180,E1 -9575.964,E2 -9575.964} C_VEL
LIN {X 0,Y 584.364,Z 584.621,A -85,B 0,C 180,E1 -9578.82,E2 -9578.82} C_VEL
LIN {X 0,Y 584.382,Z 584.619,A -85,B 0,C 180,E1 -9581.241,E2 -9581.241} C_VEL
LIN {X 0,Y 584.393,Z 584.626,A -85,B 0,C 180,E1 -9584.041,E2 -9584.041} C_VEL
LIN {X 0,Y 584.395,Z 584.617,A -85,B 0,C 180,E1 -9586.981,E2 -9586.981} C_VEL
LIN {X 0,Y 584.41,Z 584.62,A -85,B 0,C 180,E1 -9589.668,E2 -9589.668} C_VEL
LIN {X 0,Y 584.381,Z 584.623,A -85,B 0,C 180,E1 -9592.317,E2 -9592.317} C_VEL
LIN {X 0,Y 584.435,Z 584.612,A -85,B 0,C 180,E1 -9594.881,E2 -9594.881} C_VEL
LIN {X 0,Y 584.384,Z 584.623,A -85,B 0,C 180,E1 -9597.984,E2 -9597.984} C_VEL
LIN {X 0,Y 584.403,Z 584.617,A -85,B 0,C 180,E1 -9600.566,E2 -9600.566} C_VEL
LIN {X 0,Y 584.415,Z 584.614,A -85,B 0,C 180,E1 -9600.98,E2 -9600.98} C_VEL
LIN {X 0,Y 583.776,Z 584.699,A -85,B 0,C 180,E1 -9601.555,E2 -9601.555} C_VEL
LIN {X 0,Y 580.91,Z 585.057,A -85,B 0,C 180,E1 -9602.487,E2 -9602.487} C_VEL
LIN {X 0,Y 578.464,Z 585.364,A -85,B 0,C 180,E1 -9603.237,E2 -9603.237} C_VEL
LIN {X 0,Y 577.406,Z 585.496,A -85,B 0,C 180,E1 -9603.816,E2 -9603.816} C_VEL
LIN {X 0,Y 577.317,Z 585.507,A -85,B 0,C 180,E1 -9604.013,E2 -9604.013} C_VEL
LIN {X 0,Y 577.367,Z 585.496,A -85,B 0,C 180,E1 -9606.4,E2 -9606.4} C_VEL
LIN {X 0,Y 577.387,Z 585.492,A -85,B 0,C 180,E1 -9609.402,E2 -9609.402} C_VEL
LIN {X 0,Y 577.365,Z 585.497,A -85,B 0,C 180,E1 -9612.344,E2 -9612.344} C_VEL
LIN {X 0,Y 577.427,Z 585.486,A -85,B 0,C 180,E1 -9615.242,E2 -9615.242} C_VEL
LIN {X 0,Y 577.424,Z 585.487,A -85,B 0,C 180,E1 -9617.388,E2 -9617.388} C_VEL
LIN {X 0,Y 577.43,Z 585.49,A -85,B 0,C 180,E1 -9620.222,E2 -9620.222} C_VEL
LIN {X 0,Y 577.488,Z 585.477,A -85,B 0,C 180,E1 -9623.033,E2 -9623.033} C_VEL
LIN {X 0,Y 577.539,Z 585.479,A -85,B 0,C 180,E1 -9625.827,E2 -9625.827} C_VEL
LIN {X 0,Y 577.667,Z 585.456,A -85,B 0,C 180,E1 -9629.305,E2 -9629.305} C_VEL
LIN {X 0,Y 577.574,Z 585.469,A -85,B 0,C 180,E1 -9631.39,E2 -9631.39} C_VEL
LIN {X 0,Y 577.568,Z 585.467,A -85,B 0,C 180,E1 -9634.87,E2 -9634.87} C_VEL
LIN {X 0,Y 577.473,Z 585.484,A -85,B 0,C 180,E1 -9637.667,E2 -9637.667} C_VEL
LIN {X 0,Y 577.441,Z 585.484,A -85,B 0,C 180,E1 -9640.725,E2 -9640.725} C_VEL
LIN {X 0,Y 577.432,Z 585.486,A -85,B 0,C 180,E1 -9643.325,E2 -9643.325} C_VEL
LIN {X 0,Y 577.401,Z 585.494,A -85,B 0,C 180,E1 -9646.201,E2 -9646.201} C_VEL
LIN {X 0,Y 577.372,Z 585.492,A -85,B 0,C 180,E1 -9649.12,E2 -9649.12} C_VEL
LIN {X 0,Y 577.394,Z 585.491,A -85,B 0,C 180,E1 -9651.342,E2 -9651.342} C_VEL
LIN {X 0,Y 577.388,Z 585.494,A -85,B 0,C 180,E1 -9654.36,E2 -9654.36} C_VEL
LIN {X 0,Y 577.362,Z 585.498,A -85,B 0,C 180,E1 -9657.673,E2 -9657.673} C_VEL
LIN {X 0,Y 577.38,Z 585.499,A -85,B 0,C 180,E1 -9659.827,E2 -9659.827} C_VEL
LIN {X 0,Y 577.342,Z 585.501,A -85,B 0,C 180,E1 -9662.264,E2 -9662.264} C_VEL
LIN {X 0,Y 577.372,Z 585.492,A -85,B 0,C 180,E1 -9664.763,E2 -9664.763} C_VEL
LIN {X 0,Y 577.384,Z 585.492,A -85,B 0,C 180,E1 -9667.342,E2 -9667.342} C_VEL
LIN {X 0,Y 577.369,Z 585.499,A -85,B 0,C 180,E1 -9670.157,E2 -9670.157} C_VEL
LIN {X 0,Y 577.344,Z 585.496,A -85,B 0,C 180,E1 -9672.797,E2 -9672.797} C_VEL
LIN {X 0,Y 577.356,Z 585.5,A -85,B 0,C 180,E1 -9675.707,E2 -9675.707} C_VEL
LIN {X 0,Y 577.349,Z 585.502,A -85,B 0,C 180,E1 -9678.144,E2 -9678.144} C_VEL
LIN {X 0,Y 577.316,Z 585.499,A -85,B 0,C 180,E1 -9680.884,E2 -9680.884} C_VEL
LIN {X 0,Y 577.383,Z 585.494,A -85,B 0,C 180,E1 -9683.528,E2 -9683.528} C_VEL
LIN {X 0,Y 577.34,Z 585.504,A -85,B 0,C 180,E1 -9686.077,E2 -9686.077} C_VEL
LIN {X 0,Y 577.351,Z 585.496,A -85,B 0,C 180,E1 -9688.556,E2 -9688.556} C_VEL
LIN {X 0,Y 577.386,Z 585.49,A -85,B 0,C 180,E1 -9690.971,E2 -9690.971} C_VEL
LIN {X 0,Y 577.326,Z 585.506,A -85,B 0,C 180,E1 -9693.872,E2 -9693.872} C_VEL
LIN {X 0,Y 577.369,Z 585.495,A -85,B 0,C 180,E1 -9696.401,E2 -9696.401} C_VEL
LIN {X 0,Y 577.39,Z 585.492,A -85,B 0,C 180,E1 -9699.403,E2 -9699.403} C_VEL
LIN {X 0,Y 577.335,Z 585.5,A -85,B 0,C 180,E1 -9702.344,E2 -9702.344} C_VEL
LIN {X 0,Y 577.42,Z 585.487,A -85,B 0,C 180,E1 -9705.242,E2 -9705.242} C_VEL
LIN {X 0,Y 577.392,Z 585.497,A -85,B 0,C 180,E1 -9708.099,E2 -9708.099} C_VEL
LIN {X 0,Y 577.443,Z 585.489,A -85,B 0,C 180,E1 -9710.223,E2 -9710.223} C_VEL
LIN {X 0,Y 577.492,Z 585.477,A -85,B 0,C 180,E1 -9713.034,E2 -9713.034} C_VEL
LIN {X 0,Y 577.549,Z 585.47,A -85,B 0,C 180,E1 -9715.13,E2 -9715.13} C_VEL
LIN {X 0,Y 577.657,Z 585.458,A -85,B 0,C 180,E1 -9719.305,E2 -9719.305} C_VEL
LIN {X 0,Y 577.565,Z 585.47,A -85,B 0,C 180,E1 -9721.39,E2 -9721.39} C_VEL
LIN {X 0,Y 577.554,Z 585.469,A -85,B 0,C 180,E1 -9724.87,E2 -9724.87} C_VEL
LIN {X 0,Y 577.492,Z 585.477,A -85,B 0,C 180,E1 -9726.967,E2 -9726.967} C_VEL
LIN {X 0,Y 577.444,Z 585.49,A -85,B 0,C 180,E1 -9729.778,E2 -9729.778} C_VEL
LIN {X 0,Y 577.385,Z 585.491,A -85,B 0,C 180,E1 -9732.613,E2 -9732.613} C_VEL
LIN {X 0,Y 577.375,Z 585.492,A -85,B 0,C 180,E1 -9734.76,E2 -9734.76} C_VEL
LIN {X 0,Y 577.335,Z 585.497,A -85,B 0,C 180,E1 -9736.929,E2 -9736.929} C_VEL
LIN {X 0,Y 577.358,Z 585.494,A -85,B 0,C 180,E1 -9739.121,E2 -9739.121} C_VEL
LIN {X 0,Y 577.366,Z 585.5,A -85,B 0,C 180,E1 -9742.091,E2 -9742.091} C_VEL
LIN {X 0,Y 577.364,Z 585.495,A -85,B 0,C 180,E1 -9744.511,E2 -9744.511} C_VEL
LIN {X 0,Y 577.364,Z 585.498,A -85,B 0,C 180,E1 -9747.672,E2 -9747.672} C_VEL
LIN {X 0,Y 577.334,Z 585.505,A -85,B 0,C 180,E1 -9749.83,E2 -9749.83} C_VEL
LIN {X 0,Y 577.314,Z 585.504,A -85,B 0,C 180,E1 -9752.266,E2 -9752.266} C_VEL
LIN {X 0,Y 577.329,Z 585.498,A -85,B 0,C 180,E1 -9754.766,E2 -9754.766} C_VEL
LIN {X 0,Y 577.315,Z 585.501,A -85,B 0,C 180,E1 -9757.347,E2 -9757.347} C_VEL
LIN {X 0,Y 577.324,Z 585.505,A -85,B 0,C 180,E1 -9760.151,E2 -9760.151} C_VEL
LIN {X 0,Y 577.338,Z 585.496,A -85,B 0,C 180,E1 -9762.797,E2 -9762.797} C_VEL
LIN {X 0,Y 577.358,Z 585.5,A -85,B 0,C 180,E1 -9765.707,E2 -9765.707} C_VEL
LIN {X 0,Y 577.328,Z 585.504,A -85,B 0,C 180,E1 -9768.142,E2 -9768.142} C_VEL
LIN {X 0,Y 577.311,Z 585.499,A -85,B 0,C 180,E1 -9770.941,E2 -9770.941} C_VEL
LIN {X 0,Y 577.328,Z 585.501,A -85,B 0,C 180,E1 -9773.524,E2 -9773.524} C_VEL
LIN {X 0,Y 577.311,Z 585.508,A -85,B 0,C 180,E1 -9776.075,E2 -9776.075} C_VEL
LIN {X 0,Y 577.317,Z 585.5,A -85,B 0,C 180,E1 -9778.553,E2 -9778.553} C_VEL
LIN {X 0,Y 577.35,Z 585.495,A -85,B 0,C 180,E1 -9780.969,E2 -9780.969} C_VEL
LIN {X 0,Y 577.312,Z 585.501,A -85,B 0,C 180,E1 -9783.326,E2 -9783.326} C_VEL
LIN {X 0,Y 577.372,Z 585.502,A -85,B 0,C 180,E1 -9785.64,E2 -9785.64} C_VEL
LIN {X 0,Y 577.372,Z 585.641,A -85,B 0,C 180,E1 -9786.541,E2 -9786.541} C_VEL
LIN {X 0,Y 579.29,Z 596.36,A -85,B 0,C 180,E1 -9788.342,E2 -9788.342} C_VEL
LIN {X 0,Y 578.796,Z 610.137,A -85,B 0,C 180,E1 -9790.525,E2 -9790.525} C_VEL
LIN {X 0,Y 577.935,Z 630.169,A -85,B 0,C 180,E1 -9793.657,E2 -9793.657} C_VEL
LIN {X 0,Y 577.392,Z 647.603,A -85,B 0,C 180,E1 -9796.353,E2 -9796.353} C_VEL
LIN {X 0,Y 579.722,Z 666.792,A -85,B 0,C 180,E1 -9796.671,E2 -9796.671} C_VEL
LIN {X 0,Y 578.945,Z 753.769,A -85,B 0,C 180,E1 -9797.865,E2 -9797.865} C_VEL
LIN {X 0,Y 578.759,Z 764.06,A -85,B 0,C 180,E1 -9798.083,E2 -9798.083} C_VEL
LIN {X 0,Y 578.551,Z 774.272,A -85,B 0,C 180,E1 -9798.388,E2 -9798.388} C_VEL
LIN {X 0,Y 578.305,Z 783.355,A -85,B 0,C 180,E1 -9798.738,E2 -9798.738} C_VEL
LIN {X 0,Y 578.027,Z 795.028,A -85,B 0,C 180,E1 -9799.321,E2 -9799.321} C_VEL
LIN {X 0,Y 577.659,Z 804.031,A -85,B 0,C 180,E1 -9799.874,E2 -9799.874} C_VEL
LIN {X 0,Y 577.339,Z 813.415,A -85,B 0,C 180,E1 -9800.573,E2 -9800.573} C_VEL
LIN {X 0,Y 577.018,Z 821.289,A -85,B 0,C 180,E1 -9801.272,E2 -9801.272} C_VEL
LIN {X 0,Y 576.757,Z 829.476,A -85,B 0,C 180,E1 -9802.147,E2 -9802.147} C_VEL
LIN {X 0,Y 576.543,Z 836.289,A -85,B 0,C 180,E1 -9803.022,E2 -9803.022} C_VEL
LIN {X 0,Y 576.403,Z 840.993,A -85,B 0,C 180,E1 -9803.721,E2 -9803.721} C_VEL
LIN {X 0,Y 576.256,Z 846.715,A -85,B 0,C 180,E1 -9804.77,E2 -9804.77} C_VEL
LIN {X 0,Y 576.174,Z 851.212,A -85,B 0,C 180,E1 -9805.817,E2 -9805.817} C_VEL
LIN {X 0,Y 576.183,Z 853.556,A -85,B 0,C 180,E1 -9806.515,E2 -9806.515} C_VEL
LIN {X 0,Y 576.077,Z 857.009,A -85,B 0,C 180,E1 -9807.91,E2 -9807.91} C_VEL
LIN {X 0,Y 576.095,Z 858.62,A -85,B 0,C 180,E1 -9809.303,E2 -9809.303} C_VEL
LIN {X 0,Y 576.085,Z 858.926,A -85,B 0,C 180,E1 -9810,E2 -9810} C_VEL
LIN {X 0,Y 576.059,Z 858.078,A -85,B 0,C 180,E1 -9811.394,E2 -9811.394} C_VEL
LIN {X 0,Y 576.077,Z 857.079,A -85,B 0,C 180,E1 -9812.091,E2 -9812.091} C_VEL
LIN {X 0,Y 576.183,Z 853.769,A -85,B 0,C 180,E1 -9813.485,E2 -9813.485} C_VEL
LIN {X 0,Y 576.172,Z 850.044,A -85,B 0,C 180,E1 -9814.541,E2 -9814.541} C_VEL
LIN {X 0,Y 576.346,Z 845.252,A -85,B 0,C 180,E1 -9815.58,E2 -9815.58} C_VEL
LIN {X 0,Y 576.474,Z 839.127,A -85,B 0,C 180,E1 -9816.629,E2 -9816.629} C_VEL
LIN {X 0,Y 576.673,Z 832.925,A -85,B 0,C 180,E1 -9817.503,E2 -9817.503} C_VEL
LIN {X 0,Y 576.903,Z 825.448,A -85,B 0,C 180,E1 -9818.378,E2 -9818.378} C_VEL
LIN {X 0,Y 577.292,Z 816.361,A -85,B 0,C 180,E1 -9819.251,E2 -9819.251} C_VEL
LIN {X 0,Y 577.662,Z 807.635,A -85,B 0,C 180,E1 -9819.95,E2 -9819.95} C_VEL
LIN {X 0,Y 578.02,Z 798.797,A -85,B 0,C 180,E1 -9820.543,E2 -9820.543} C_VEL
LIN {X 0,Y 578.256,Z 789.44,A -85,B 0,C 180,E1 -9821.067,E2 -9821.067} C_VEL
LIN {X 0,Y 578.569,Z 778.105,A -85,B 0,C 180,E1 -9821.567,E2 -9821.567} C_VEL
LIN {X 0,Y 578.777,Z 767.874,A -85,B 0,C 180,E1 -9821.917,E2 -9821.917} C_VEL
LIN {X 0,Y 579.132,Z 756.226,A -85,B 0,C 180,E1 -9822.198,E2 -9822.198} C_VEL
LIN {X 0,Y 579.336,Z 735.979,A -85,B 0,C 180,E1 -9822.503,E2 -9822.503} C_VEL
LIN {X 0,Y 579.987,Z 665.674,A -85,B 0,C 180,E1 -9823.49,E2 -9823.49} C_VEL
LIN {X 0,Y 577.669,Z 648.455,A -85,B 0,C 180,E1 -9823.807,E2 -9823.807} C_VEL
LIN {X 0,Y 577.46,Z 646.852,A -85,B 0,C 180,E1 -9823.845,E2 -9823.845} C_VEL
LIN {X 0,Y 578.072,Z 629.84,A -85,B 0,C 180,E1 -9826.512,E2 -9826.512} C_VEL
LIN {X 0,Y 578.954,Z 611.187,A -85,B 0,C 180,E1 -9829.49,E2 -9829.49} C_VEL
LIN {X 0,Y 579.557,Z 597.836,A -85,B 0,C 180,E1 -9831.677,E2 -9831.677} C_VEL
LIN {X 0,Y 577.66,Z 587.104,A -85,B 0,C 180,E1 -9833.587,E2 -9833.587} C_VEL
LIN {X 0,Y 577.352,Z 585.505,A -85,B 0,C 180,E1 -9833.885,E2 -9833.885} C_VEL
LIN {X 0,Y 577.314,Z 585.508,A -85,B 0,C 180,E1 -9836.674,E2 -9836.674} C_VEL
LIN {X 0,Y 577.33,Z 585.507,A -85,B 0,C 180,E1 -9839.128,E2 -9839.128} C_VEL
LIN {X 0,Y 577.315,Z 585.505,A -85,B 0,C 180,E1 -9842.266,E2 -9842.266} C_VEL
LIN {X 0,Y 577.355,Z 585.496,A -85,B 0,C 180,E1 -9844.765,E2 -9844.765} C_VEL
LIN {X 0,Y 577.331,Z 585.502,A -85,B 0,C 180,E1 -9847.346,E2 -9847.346} C_VEL
LIN {X 0,Y 577.33,Z 585.497,A -85,B 0,C 180,E1 -9850.151,E2 -9850.151} C_VEL
LIN {X 0,Y 577.345,Z 585.497,A -85,B 0,C 180,E1 -9852.797,E2 -9852.797} C_VEL
LIN {X 0,Y 577.361,Z 585.499,A -85,B 0,C 180,E1 -9855.707,E2 -9855.707} C_VEL
LIN {X 0,Y 577.354,Z 585.497,A -85,B 0,C 180,E1 -9858.144,E2 -9858.144} C_VEL
LIN {X 0,Y 577.317,Z 585.506,A -85,B 0,C 180,E1 -9860.883,E2 -9860.883} C_VEL
LIN {X 0,Y 577.388,Z 585.495,A -85,B 0,C 180,E1 -9863.528,E2 -9863.528} C_VEL
LIN {X 0,Y 577.347,Z 585.497,A -85,B 0,C 180,E1 -9866.077,E2 -9866.077} C_VEL
LIN {X 0,Y 577.354,Z 585.5,A -85,B 0,C 180,E1 -9868.555,E2 -9868.555} C_VEL
LIN {X 0,Y 577.39,Z 585.497,A -85,B 0,C 180,E1 -9870.971,E2 -9870.971} C_VEL
LIN {X 0,Y 577.315,Z 585.503,A -85,B 0,C 180,E1 -9873.874,E2 -9873.874} C_VEL
LIN {X 0,Y 577.373,Z 585.5,A -85,B 0,C 180,E1 -9876.4,E2 -9876.4} C_VEL
LIN {X 0,Y 577.394,Z 585.495,A -85,B 0,C 180,E1 -9879.402,E2 -9879.402} C_VEL
LIN {X 0,Y 577.365,Z 585.506,A -85,B 0,C 180,E1 -9882.344,E2 -9882.344} C_VEL
LIN {X 0,Y 577.424,Z 585.491,A -85,B 0,C 180,E1 -9885.242,E2 -9885.242} C_VEL
LIN {X 0,Y 577.396,Z 585.498,A -85,B 0,C 180,E1 -9888.098,E2 -9888.098} C_VEL
LIN {X 0,Y 577.462,Z 585.668,A -85,B 0,C 180,E1 -9888.975,E2 -9888.975} C_VEL
LIN {X 0,Y 578.82,Z 593.612,A -85,B 0,C 180,E1 -9890.597,E2 -9890.597} C_VEL
LIN {X 0,Y 578.795,Z 600.906,A -85,B 0,C 180,E1 -9892,E2 -9892} C_VEL
LIN {X 0,Y 577.987,Z 617.698,A -85,B 0,C 180,E1 -9895.134,E2 -9895.134} C_VEL
LIN {X 0,Y 577.596,Z 623.612,A -85,B 0,C 180,E1 -9896.219,E2 -9896.219} C_VEL
LIN {X 0,Y 580.278,Z 639.695,A -85,B 0,C 180,E1 -9896.54,E2 -9896.54} C_VEL
LIN {X 0,Y 579.036,Z 729.63,A -85,B 0,C 180,E1 -9897.812,E2 -9897.812} C_VEL
LIN {X 0,Y 578.861,Z 739.352,A -85,B 0,C 180,E1 -9898.028,E2 -9898.028} C_VEL
LIN {X 0,Y 578.696,Z 748.631,A -85,B 0,C 180,E1 -9898.309,E2 -9898.309} C_VEL
LIN {X 0,Y 578.498,Z 758.54,A -85,B 0,C 180,E1 -9898.699,E2 -9898.699} C_VEL
LIN {X 0,Y 578.323,Z 768.907,A -85,B 0,C 180,E1 -9899.219,E2 -9899.219} C_VEL
LIN {X 0,Y 578.003,Z 778.723,A -85,B 0,C 180,E1 -9899.826,E2 -9899.826} C_VEL
LIN {X 0,Y 577.683,Z 787.955,A -85,B 0,C 180,E1 -9900.521,E2 -9900.521} C_VEL
LIN {X 0,Y 577.281,Z 795.753,A -85,B 0,C 180,E1 -9901.216,E2 -9901.216} C_VEL
LIN {X 0,Y 576.983,Z 803.844,A -85,B 0,C 180,E1 -9902.087,E2 -9902.087} C_VEL
LIN {X 0,Y 576.7,Z 810.613,A -85,B 0,C 180,E1 -9902.959,E2 -9902.959} C_VEL
LIN {X 0,Y 576.465,Z 816.272,A -85,B 0,C 180,E1 -9903.832,E2 -9903.832} C_VEL
LIN {X 0,Y 576.367,Z 821.746,A -85,B 0,C 180,E1 -9904.88,E2 -9904.88} C_VEL
LIN {X 0,Y 576.25,Z 826.046,A -85,B 0,C 180,E1 -9905.93,E2 -9905.93} C_VEL
LIN {X 0,Y 576.143,Z 829.273,A -85,B 0,C 180,E1 -9906.983,E2 -9906.983} C_VEL
LIN {X 0,Y 576.044,Z 830.923,A -85,B 0,C 180,E1 -9907.686,E2 -9907.686} C_VEL
LIN {X 0,Y 576.035,Z 832.763,A -85,B 0,C 180,E1 -9909.095,E2 -9909.095} C_VEL
LIN {X 0,Y 576.094,Z 833.136,A -85,B 0,C 180,E1 -9909.989,E2 -9909.989} C_VEL
LIN {X 0,Y 576.035,Z 832.456,A -85,B 0,C 180,E1 -9911.218,E2 -9911.218} C_VEL
LIN {X 0,Y 576.013,Z 831.443,A -85,B 0,C 180,E1 -9911.93,E2 -9911.93} C_VEL
LIN {X 0,Y 576.146,Z 828.239,A -85,B 0,C 180,E1 -9913.355,E2 -9913.355} C_VEL
LIN {X 0,Y 576.221,Z 824.531,A -85,B 0,C 180,E1 -9914.43,E2 -9914.43} C_VEL
LIN {X 0,Y 576.391,Z 819.608,A -85,B 0,C 180,E1 -9915.506,E2 -9915.506} C_VEL
LIN {X 0,Y 576.543,Z 813.541,A -85,B 0,C 180,E1 -9916.552,E2 -9916.552} C_VEL
LIN {X 0,Y 576.735,Z 806.838,A -85,B 0,C 180,E1 -9917.493,E2 -9917.493} C_VEL
LIN {X 0,Y 577.046,Z 798.998,A -85,B 0,C 180,E1 -9918.397,E2 -9918.397} C_VEL
LIN {X 0,Y 577.337,Z 791.523,A -85,B 0,C 180,E1 -9919.121,E2 -9919.121} C_VEL
LIN {X 0,Y 577.585,Z 782.543,A -85,B 0,C 180,E1 -9919.85,E2 -9919.85} C_VEL
LIN {X 0,Y 577.926,Z 773.063,A -85,B 0,C 180,E1 -9920.485,E2 -9920.485} C_VEL
LIN {X 0,Y 578.273,Z 762.981,A -85,B 0,C 180,E1 -9921.036,E2 -9921.036} C_VEL
LIN {X 0,Y 578.488,Z 752.711,A -85,B 0,C 180,E1 -9921.486,E2 -9921.486} C_VEL
LIN {X 0,Y 578.619,Z 741.763,A -85,B 0,C 180,E1 -9921.854,E2 -9921.854} C_VEL
LIN {X 0,Y 578.902,Z 731.623,A -85,B 0,C 180,E1 -9922.099,E2 -9922.099} C_VEL
LIN {X 0,Y 579.134,Z 713.621,A -85,B 0,C 180,E1 -9922.371,E2 -9922.371} C_VEL
LIN {X 0,Y 579.795,Z 638.113,A -85,B 0,C 180,E1 -9923.404,E2 -9923.404} C_VEL
LIN {X 0,Y 577.457,Z 622.65,A -85,B 0,C 180,E1 -9923.69,E2 -9923.69} C_VEL
LIN {X 0,Y 578.036,Z 605.149,A -85,B 0,C 180,E1 -9926.832,E2 -9926.832} C_VEL
LIN {X 0,Y 578.43,Z 593.366,A -85,B 0,C 180,E1 -9928.971,E2 -9928.971} C_VEL
LIN {X 0,Y 577.455,Z 585.49,A -85,B 0,C 180,E1 -9930.48,E2 -9930.48} C_VEL
LIN {X 0,Y 577.366,Z 585.502,A -85,B 0,C 180,E1 -9933.921,E2 -9933.921} C_VEL
LIN {X 0,Y 577.383,Z 585.491,A -85,B 0,C 180,E1 -9936.806,E2 -9936.806} C_VEL
LIN {X 0,Y 577.371,Z 585.499,A -85,B 0,C 180,E1 -9940.156,E2 -9940.156} C_VEL
LIN {X 0,Y 577.346,Z 585.495,A -85,B 0,C 180,E1 -9942.796,E2 -9942.796} C_VEL
LIN {X 0,Y 577.358,Z 585.499,A -85,B 0,C 180,E1 -9945.707,E2 -9945.707} C_VEL
LIN {X 0,Y 577.35,Z 585.502,A -85,B 0,C 180,E1 -9948.144,E2 -9948.144} C_VEL
LIN {X 0,Y 577.313,Z 585.499,A -85,B 0,C 180,E1 -9950.883,E2 -9950.883} C_VEL
LIN {X 0,Y 577.382,Z 585.494,A -85,B 0,C 180,E1 -9953.527,E2 -9953.527} C_VEL
LIN {X 0,Y 577.339,Z 585.504,A -85,B 0,C 180,E1 -9956.076,E2 -9956.076} C_VEL
LIN {X 0,Y 577.349,Z 585.496,A -85,B 0,C 180,E1 -9958.555,E2 -9958.555} C_VEL
LIN {X 0,Y 577.384,Z 585.49,A -85,B 0,C 180,E1 -9960.973,E2 -9960.973} C_VEL
LIN {X 0,Y 577.324,Z 585.506,A -85,B 0,C 180,E1 -9963.871,E2 -9963.871} C_VEL
LIN {X 0,Y 577.317,Z 585.507,A -85,B 0,C 180,E1 -9964.013,E2 -9964.013} C_VEL
LIN {X 0,Y 576.647,Z 585.589,A -85,B 0,C 180,E1 -9964.595,E2 -9964.595} C_VEL
LIN {X 0,Y 573.81,Z 585.939,A -85,B 0,C 180,E1 -9965.541,E2 -9965.541} C_VEL
LIN {X 0,Y 571.42,Z 586.238,A -85,B 0,C 180,E1 -9966.302,E2 -9966.302} C_VEL
LIN {X 0,Y 570.399,Z 586.361,A -85,B 0,C 180,E1 -9966.889,E2 -9966.889} C_VEL
LIN {X 0,Y 570.318,Z 586.371,A -85,B 0,C 180,E1 -9967.088,E2 -9967.088} C_VEL
LIN {X 0,Y 570.316,Z 586.38,A -85,B 0,C 180,E1 -9969.886,E2 -9969.886} C_VEL
LIN {X 0,Y 570.338,Z 586.368,A -85,B 0,C 180,E1 -9972.857,E2 -9972.857} C_VEL
LIN {X 0,Y 570.387,Z 586.372,A -85,B 0,C 180,E1 -9975.959,E2 -9975.959} C_VEL
LIN {X 0,Y 570.407,Z 586.36,A -85,B 0,C 180,E1 -9979.225,E2 -9979.225} C_VEL
LIN {X 0,Y 570.441,Z 586.361,A -85,B 0,C 180,E1 -9982.237,E2 -9982.237} C_VEL
LIN {X 0,Y 570.52,Z 586.346,A -85,B 0,C 180,E1 -9985.07,E2 -9985.07} C_VEL
LIN {X 0,Y 570.643,Z 586.331,A -85,B 0,C 180,E1 -9989.297,E2 -9989.297} C_VEL
LIN {X 0,Y 570.522,Z 586.347,A -85,B 0,C 180,E1 -9991.407,E2 -9991.407} C_VEL
LIN {X 0,Y 570.519,Z 586.345,A -85,B 0,C 180,E1 -9994.93,E2 -9994.93} C_VEL
LIN {X 0,Y 570.441,Z 586.362,A -85,B 0,C 180,E1 -9997.762,E2 -9997.762} C_VEL
LIN {X 0,Y 570.407,Z 586.36,A -85,B 0,C 180,E1 -10000.775,E2 -10000.775} C_VEL
LIN {X 0,Y 570.386,Z 586.371,A -85,B 0,C 180,E1 -10004.041,E2 -10004.041} C_VEL
LIN {X 0,Y 570.338,Z 586.369,A -85,B 0,C 180,E1 -10007.142,E2 -10007.142} C_VEL
LIN {X 0,Y 570.327,Z 586.377,A -85,B 0,C 180,E1 -10010.113,E2 -10010.113} C_VEL
LIN {X 0,Y 570.318,Z 586.371,A -85,B 0,C 180,E1 -10012.911,E2 -10012.911} C_VEL
LIN {X 0,Y 570.262,Z 586.38,A -85,B 0,C 180,E1 -10015.461,E2 -10015.461} C_VEL
LIN {X 0,Y 570.327,Z 586.377,A -85,B 0,C 180,E1 -10017.84,E2 -10017.84} C_VEL
LIN {X 0,Y 570.319,Z 586.371,A -85,B 0,C 180,E1 -10020.717,E2 -10020.717} C_VEL
LIN {X 0,Y 570.337,Z 586.372,A -85,B 0,C 180,E1 -10023.549,E2 -10023.549} C_VEL
LIN {X 0,Y 570.354,Z 586.373,A -85,B 0,C 180,E1 -10026.12,E2 -10026.12} C_VEL
LIN {X 0,Y 570.279,Z 586.376,A -85,B 0,C 180,E1 -10028.785,E2 -10028.785} C_VEL
LIN {X 0,Y 570.301,Z 586.376,A -85,B 0,C 180,E1 -10031.547,E2 -10031.547} C_VEL
LIN {X 0,Y 570.307,Z 586.373,A -85,B 0,C 180,E1 -10034.574,E2 -10034.574} C_VEL
LIN {X 0,Y 570.305,Z 586.375,A -85,B 0,C 180,E1 -10037.507,E2 -10037.507} C_VEL
LIN {X 0,Y 570.289,Z 586.379,A -85,B 0,C 180,E1 -10040.307,E2 -10040.307} C_VEL
LIN {X 0,Y 570.349,Z 586.367,A -85,B 0,C 180,E1 -10043.004,E2 -10043.004} C_VEL
LIN {X 0,Y 570.314,Z 586.375,A -85,B 0,C 180,E1 -10045.601,E2 -10045.601} C_VEL
LIN {X 0,Y 570.325,Z 586.377,A -85,B 0,C 180,E1 -10048.123,E2 -10048.123} C_VEL
LIN {X 0,Y 570.314,Z 586.372,A -85,B 0,C 180,E1 -10050.692,E2 -10050.692} C_VEL
LIN {X 0,Y 570.302,Z 586.373,A -85,B 0,C 180,E1 -10052.972,E2 -10052.972} C_VEL
LIN {X 0,Y 570.332,Z 586.377,A -85,B 0,C 180,E1 -10056.091,E2 -10056.091} C_VEL
LIN {X 0,Y 570.357,Z 586.366,A -85,B 0,C 180,E1 -10059.137,E2 -10059.137} C_VEL
LIN {X 0,Y 570.313,Z 586.379,A -85,B 0,C 180,E1 -10062.119,E2 -10062.119} C_VEL
LIN {X 0,Y 570.373,Z 586.364,A -85,B 0,C 180,E1 -10065.055,E2 -10065.055} C_VEL
LIN {X 0,Y 570.366,Z 586.375,A -85,B 0,C 180,E1 -10067.95,E2 -10067.95} C_VEL
LIN {X 0,Y 570.395,Z 586.369,A -85,B 0,C 180,E1 -10070.101,E2 -10070.101} C_VEL
LIN {X 0,Y 570.441,Z 586.355,A -85,B 0,C 180,E1 -10072.947,E2 -10072.947} C_VEL
LIN {X 0,Y 570.501,Z 586.348,A -85,B 0,C 180,E1 -10075.07,E2 -10075.07} C_VEL
LIN {X 0,Y 570.635,Z 586.332,A -85,B 0,C 180,E1 -10079.297,E2 -10079.297} C_VEL
LIN {X 0,Y 570.512,Z 586.349,A -85,B 0,C 180,E1 -10081.407,E2 -10081.407} C_VEL
LIN {X 0,Y 570.506,Z 586.347,A -85,B 0,C 180,E1 -10084.93,E2 -10084.93} C_VEL
LIN {X 0,Y 570.441,Z 586.355,A -85,B 0,C 180,E1 -10087.053,E2 -10087.053} C_VEL
LIN {X 0,Y 570.395,Z 586.37,A -85,B 0,C 180,E1 -10089.9,E2 -10089.9} C_VEL
LIN {X 0,Y 570.337,Z 586.369,A -85,B 0,C 180,E1 -10092.772,E2 -10092.772} C_VEL
LIN {X 0,Y 570.325,Z 586.37,A -85,B 0,C 180,E1 -10094.946,E2 -10094.946} C_VEL
LIN {X 0,Y 570.292,Z 586.374,A -85,B 0,C 180,E1 -10097.144,E2 -10097.144} C_VEL
LIN {X 0,Y 570.292,Z 586.376,A -85,B 0,C 180,E1 -10099.367,E2 -10099.367} C_VEL
LIN {X 0,Y 570.307,Z 586.377,A -85,B 0,C 180,E1 -10101.621,E2 -10101.621} C_VEL
LIN {X 0,Y 570.318,Z 586.38,A -85,B 0,C 180,E1 -10103.91,E2 -10103.91} C_VEL
LIN {X 0,Y 570.288,Z 586.375,A -85,B 0,C 180,E1 -10107.029,E2 -10107.029} C_VEL
LIN {X 0,Y 570.296,Z 586.376,A -85,B 0,C 180,E1 -10109.425,E2 -10109.425} C_VEL
LIN {X 0,Y 570.274,Z 586.385,A -85,B 0,C 180,E1 -10112.059,E2 -10112.059} C_VEL
LIN {X 0,Y 570.28,Z 586.377,A -85,B 0,C 180,E1 -10114.621,E2 -10114.621} C_VEL
LIN {X 0,Y 570.28,Z 586.375,A -85,B 0,C 180,E1 -10117.026,E2 -10117.026} C_VEL
LIN {X 0,Y 570.277,Z 586.381,A -85,B 0,C 180,E1 -10119.694,E2 -10119.694} C_VEL
LIN {X 0,Y 570.293,Z 586.376,A -85,B 0,C 180,E1 -10122.529,E2 -10122.529} C_VEL
LIN {X 0,Y 570.309,Z 586.376,A -85,B 0,C 180,E1 -10125.568,E2 -10125.568} C_VEL
LIN {X 0,Y 570.269,Z 586.379,A -85,B 0,C 180,E1 -10128.525,E2 -10128.525} C_VEL
LIN {X 0,Y 570.26,Z 586.379,A -85,B 0,C 180,E1 -10131.213,E2 -10131.213} C_VEL
LIN {X 0,Y 570.303,Z 586.379,A -85,B 0,C 180,E1 -10134.155,E2 -10134.155} C_VEL
LIN {X 0,Y 570.273,Z 586.377,A -85,B 0,C 180,E1 -10136.638,E2 -10136.638} C_VEL
LIN {X 0,Y 570.272,Z 586.378,A -85,B 0,C 180,E1 -10139.292,E2 -10139.292} C_VEL
LIN {X 0,Y 570.29,Z 586.38,A -85,B 0,C 180,E1 -10142.178,E2 -10142.178} C_VEL
LIN {X 0,Y 570.311,Z 586.378,A -85,B 0,C 180,E1 -10145.347,E2 -10145.347} C_VEL
LIN {X 0,Y 570.333,Z 586.547,A -85,B 0,C 180,E1 -10146.428,E2 -10146.428} C_VEL
LIN {X 0,Y 572.296,Z 597.482,A -85,B 0,C 180,E1 -10148.289,E2 -10148.289} C_VEL
LIN {X 0,Y 571.746,Z 612.022,A -85,B 0,C 180,E1 -10150.617,E2 -10150.617} C_VEL
LIN {X 0,Y 570.881,Z 632.09,A -85,B 0,C 180,E1 -10153.792,E2 -10153.792} C_VEL
LIN {X 0,Y 570.345,Z 647.565,A -85,B 0,C 180,E1 -10156.203,E2 -10156.203} C_VEL
LIN {X 0,Y 572.765,Z 667.224,A -85,B 0,C 180,E1 -10156.532,E2 -10156.532} C_VEL
LIN {X 0,Y 571.945,Z 754.408,A -85,B 0,C 180,E1 -10157.759,E2 -10157.759} C_VEL
LIN {X 0,Y 571.736,Z 764.402,A -85,B 0,C 180,E1 -10157.979,E2 -10157.979} C_VEL
LIN {X 0,Y 571.525,Z 774.472,A -85,B 0,C 180,E1 -10158.289,E2 -10158.289} C_VEL
LIN {X 0,Y 571.252,Z 784.404,A -85,B 0,C 180,E1 -10158.686,E2 -10158.686} C_VEL
LIN {X 0,Y 571.031,Z 793.969,A -85,B 0,C 180,E1 -10159.167,E2 -10159.167} C_VEL
LIN {X 0,Y 570.65,Z 803.444,A -85,B 0,C 180,E1 -10159.748,E2 -10159.748} C_VEL
LIN {X 0,Y 570.323,Z 812.907,A -85,B 0,C 180,E1 -10160.456,E2 -10160.456} C_VEL
LIN {X 0,Y 569.967,Z 820.844,A -85,B 0,C 180,E1 -10161.164,E2 -10161.164} C_VEL
LIN {X 0,Y 569.708,Z 829.087,A -85,B 0,C 180,E1 -10162.05,E2 -10162.05} C_VEL
LIN {X 0,Y 569.454,Z 835.945,A -85,B 0,C 180,E1 -10162.935,E2 -10162.935} C_VEL
LIN {X 0,Y 569.323,Z 840.675,A -85,B 0,C 180,E1 -10163.643,E2 -10163.643} C_VEL
LIN {X 0,Y 569.178,Z 846.444,A -85,B 0,C 180,E1 -10164.704,E2 -10164.704} C_VEL
LIN {X 0,Y 569.089,Z 850.974,A -85,B 0,C 180,E1 -10165.765,E2 -10165.765} C_VEL
LIN {X 0,Y 569.081,Z 853.319,A -85,B 0,C 180,E1 -10166.472,E2 -10166.472} C_VEL
LIN {X 0,Y 568.996,Z 856.815,A -85,B 0,C 180,E1 -10167.884,E2 -10167.884} C_VEL
LIN {X 0,Y 568.998,Z 858.45,A -85,B 0,C 180,E1 -10169.295,E2 -10169.295} C_VEL
LIN {X 0,Y 568.987,Z 858.76,A -85,B 0,C 180,E1 -10170,E2 -10170} C_VEL
LIN {X 0,Y 568.97,Z 857.938,A -85,B 0,C 180,E1 -10171.411,E2 -10171.411} C_VEL
LIN {X 0,Y 568.997,Z 856.935,A -85,B 0,C 180,E1 -10172.117,E2 -10172.117} C_VEL
LIN {X 0,Y 569.081,Z 853.646,A -85,B 0,C 180,E1 -10173.528,E2 -10173.528} C_VEL
LIN {X 0,Y 569.095,Z 849.457,A -85,B 0,C 180,E1 -10174.704,E2 -10174.704} C_VEL
LIN {X 0,Y 569.266,Z 845.137,A -85,B 0,C 180,E1 -10175.649,E2 -10175.649} C_VEL
LIN {X 0,Y 569.421,Z 839.024,A -85,B 0,C 180,E1 -10176.711,E2 -10176.711} C_VEL
LIN {X 0,Y 569.611,Z 832.841,A -85,B 0,C 180,E1 -10177.596,E2 -10177.596} C_VEL
LIN {X 0,Y 569.857,Z 825.39,A -85,B 0,C 180,E1 -10178.482,E2 -10178.482} C_VEL
LIN {X 0,Y 570.296,Z 816.341,A -85,B 0,C 180,E1 -10179.366,E2 -10179.366} C_VEL
LIN {X 0,Y 570.683,Z 807.646,A -85,B 0,C 180,E1 -10180.073,E2 -10180.073} C_VEL
LIN {X 0,Y 571.046,Z 797.956,A -85,B 0,C 180,E1 -10180.726,E2 -10180.726} C_VEL
LIN {X 0,Y 571.324,Z 788.629,A -85,B 0,C 180,E1 -10181.246,E2 -10181.246} C_VEL
LIN {X 0,Y 571.623,Z 778.268,A -85,B 0,C 180,E1 -10181.71,E2 -10181.71} C_VEL
LIN {X 0,Y 571.886,Z 767.358,A -85,B 0,C 180,E1 -10182.085,E2 -10182.085} C_VEL
LIN {X 0,Y 572.212,Z 756.789,A -85,B 0,C 180,E1 -10182.347,E2 -10182.347} C_VEL
LIN {X 0,Y 572.437,Z 736.828,A -85,B 0,C 180,E1 -10182.657,E2 -10182.657} C_VEL
LIN {X 0,Y 573.129,Z 666.288,A -85,B 0,C 180,E1 -10183.667,E2 -10183.667} C_VEL
LIN {X 0,Y 571.095,Z 650.639,A -85,B 0,C 180,E1 -10183.963,E2 -10183.963} C_VEL
LIN {X 0,Y 570.501,Z 646.609,A -85,B 0,C 180,E1 -10184.059,E2 -10184.059} C_VEL
LIN {X 0,Y 571.322,Z 626.321,A -85,B 0,C 180,E1 -10187.296,E2 -10187.296} C_VEL
LIN {X 0,Y 572.219,Z 608.331,A -85,B 0,C 180,E1 -10190.231,E2 -10190.231} C_VEL
LIN {X 0,Y 572.629,Z 599.982,A -85,B 0,C 180,E1 -10191.622,E2 -10191.622} C_VEL
LIN {X 0,Y 571.772,Z 593.923,A -85,B 0,C 180,E1 -10192.699,E2 -10192.699} C_VEL
LIN {X 0,Y 570.315,Z 586.381,A -85,B 0,C 180,E1 -10194.102,E2 -10194.102} C_VEL
LIN {X 0,Y 570.281,Z 586.385,A -85,B 0,C 180,E1 -10197.03,E2 -10197.03} C_VEL
LIN {X 0,Y 570.289,Z 586.384,A -85,B 0,C 180,E1 -10199.426,E2 -10199.426} C_VEL
LIN {X 0,Y 570.274,Z 586.384,A -85,B 0,C 180,E1 -10202.06,E2 -10202.06} C_VEL
LIN {X 0,Y 570.323,Z 586.372,A -85,B 0,C 180,E1 -10204.628,E2 -10204.628} C_VEL
LIN {X 0,Y 570.318,Z 586.374,A -85,B 0,C 180,E1 -10207.031,E2 -10207.031} C_VEL
LIN {X 0,Y 570.28,Z 586.377,A -85,B 0,C 180,E1 -10209.694,E2 -10209.694} C_VEL
LIN {X 0,Y 570.298,Z 586.373,A -85,B 0,C 180,E1 -10212.53,E2 -10212.53} C_VEL
LIN {X 0,Y 570.313,Z 586.379,A -85,B 0,C 180,E1 -10215.568,E2 -10215.568} C_VEL
LIN {X 0,Y 570.305,Z 586.377,A -85,B 0,C 180,E1 -10218.521,E2 -10218.521} C_VEL
LIN {X 0,Y 570.271,Z 586.385,A -85,B 0,C 180,E1 -10221.214,E2 -10221.214} C_VEL
LIN {X 0,Y 570.369,Z 586.367,A -85,B 0,C 180,E1 -10224.147,E2 -10224.147} C_VEL
LIN {X 0,Y 570.315,Z 586.377,A -85,B 0,C 180,E1 -10226.633,E2 -10226.633} C_VEL
LIN {X 0,Y 570.307,Z 586.376,A -85,B 0,C 180,E1 -10229.287,E2 -10229.287} C_VEL
LIN {X 0,Y 570.33,Z 586.374,A -85,B 0,C 180,E1 -10232.18,E2 -10232.18} C_VEL
LIN {X 0,Y 570.319,Z 586.375,A -85,B 0,C 180,E1 -10235.346,E2 -10235.346} C_VEL
LIN {X 0,Y 570.324,Z 586.376,A -85,B 0,C 180,E1 -10237.621,E2 -10237.621} C_VEL
LIN {X 0,Y 570.322,Z 586.378,A -85,B 0,C 180,E1 -10239.886,E2 -10239.886} C_VEL
LIN {X 0,Y 570.334,Z 586.38,A -85,B 0,C 180,E1 -10242.119,E2 -10242.119} C_VEL
LIN {X 0,Y 570.377,Z 586.37,A -85,B 0,C 180,E1 -10245.055,E2 -10245.055} C_VEL
LIN {X 0,Y 570.37,Z 586.373,A -85,B 0,C 180,E1 -10247.95,E2 -10247.95} C_VEL
LIN {X 0,Y 570.393,Z 586.428,A -85,B 0,C 180,E1 -10248.749,E2 -10248.749} C_VEL
LIN {X 0,Y 571.853,Z 594.752,A -85,B 0,C 180,E1 -10250.482,E2 -10250.482} C_VEL
LIN {X 0,Y 571.853,Z 602.003,A -85,B 0,C 180,E1 -10251.902,E2 -10251.902} C_VEL
LIN {X 0,Y 571.041,Z 616.908,A -85,B 0,C 180,E1 -10254.721,E2 -10254.721} C_VEL
LIN {X 0,Y 570.645,Z 623.89,A -85,B 0,C 180,E1 -10256.019,E2 -10256.019} C_VEL
LIN {X 0,Y 573.395,Z 639.646,A -85,B 0,C 180,E1 -10256.345,E2 -10256.345} C_VEL
LIN {X 0,Y 572.412,Z 709.905,A -85,B 0,C 180,E1 -10257.348,E2 -10257.348} C_VEL
LIN {X 0,Y 572.099,Z 731.297,A -85,B 0,C 180,E1 -10257.675,E2 -10257.675} C_VEL
LIN {X 0,Y 571.912,Z 742.075,A -85,B 0,C 180,E1 -10257.938,E2 -10257.938} C_VEL
LIN {X 0,Y 571.706,Z 752.44,A -85,B 0,C 180,E1 -10258.288,E2 -10258.288} C_VEL
LIN {X 0,Y 571.545,Z 761.533,A -85,B 0,C 180,E1 -10258.683,E2 -10258.683} C_VEL
LIN {X 0,Y 571.35,Z 769.898,A -85,B 0,C 180,E1 -10259.122,E2 -10259.122} C_VEL
LIN {X 0,Y 571.069,Z 778.355,A -85,B 0,C 180,E1 -10259.648,E2 -10259.648} C_VEL
LIN {X 0,Y 570.743,Z 787.679,A -85,B 0,C 180,E1 -10260.351,E2 -10260.351} C_VEL
LIN {X 0,Y 570.335,Z 795.554,A -85,B 0,C 180,E1 -10261.055,E2 -10261.055} C_VEL
LIN {X 0,Y 569.943,Z 803.724,A -85,B 0,C 180,E1 -10261.937,E2 -10261.937} C_VEL
LIN {X 0,Y 569.693,Z 810.526,A -85,B 0,C 180,E1 -10262.819,E2 -10262.819} C_VEL
LIN {X 0,Y 569.405,Z 815.236,A -85,B 0,C 180,E1 -10263.526,E2 -10263.526} C_VEL
LIN {X 0,Y 569.31,Z 821.645,A -85,B 0,C 180,E1 -10264.741,E2 -10264.741} C_VEL
LIN {X 0,Y 569.188,Z 826.046,A -85,B 0,C 180,E1 -10265.818,E2 -10265.818} C_VEL
LIN {X 0,Y 569.032,Z 829.757,A -85,B 0,C 180,E1 -10267.07,E2 -10267.07} C_VEL
LIN {X 0,Y 568.944,Z 831.356,A -85,B 0,C 180,E1 -10267.783,E2 -10267.783} C_VEL
LIN {X 0,Y 568.95,Z 832.988,A -85,B 0,C 180,E1 -10269.209,E2 -10269.209} C_VEL
LIN {X 0,Y 568.995,Z 833.297,A -85,B 0,C 180,E1 -10269.996,E2 -10269.996} C_VEL
LIN {X 0,Y 568.926,Z 832.413,A -85,B 0,C 180,E1 -10271.361,E2 -10271.361} C_VEL
LIN {X 0,Y 568.929,Z 831.394,A -85,B 0,C 180,E1 -10272.081,E2 -10272.081} C_VEL
LIN {X 0,Y 569.091,Z 827.906,A -85,B 0,C 180,E1 -10273.524,E2 -10273.524} C_VEL
LIN {X 0,Y 569.174,Z 824.031,A -85,B 0,C 180,E1 -10274.612,E2 -10274.612} C_VEL
LIN {X 0,Y 569.333,Z 818.924,A -85,B 0,C 180,E1 -10275.703,E2 -10275.703} C_VEL
LIN {X 0,Y 569.471,Z 813.636,A -85,B 0,C 180,E1 -10276.617,E2 -10276.617} C_VEL
LIN {X 0,Y 569.67,Z 807.209,A -85,B 0,C 180,E1 -10277.532,E2 -10277.532} C_VEL
LIN {X 0,Y 569.976,Z 799.4,A -85,B 0,C 180,E1 -10278.448,E2 -10278.448} C_VEL
LIN {X 0,Y 570.288,Z 791.507,A -85,B 0,C 180,E1 -10279.221,E2 -10279.221} C_VEL
LIN {X 0,Y 570.563,Z 783.05,A -85,B 0,C 180,E1 -10279.917,E2 -10279.917} C_VEL
LIN {X 0,Y 570.901,Z 773.638,A -85,B 0,C 180,E1 -10280.561,E2 -10280.561} C_VEL
LIN {X 0,Y 571.267,Z 763.337,A -85,B 0,C 180,E1 -10281.133,E2 -10281.133} C_VEL
LIN {X 0,Y 571.482,Z 753.543,A -85,B 0,C 180,E1 -10281.573,E2 -10281.573} C_VEL
LIN {X 0,Y 571.646,Z 742.875,A -85,B 0,C 180,E1 -10281.945,E2 -10281.945} C_VEL
LIN {X 0,Y 571.907,Z 731.916,A -85,B 0,C 180,E1 -10282.218,E2 -10282.218} C_VEL
LIN {X 0,Y 572.142,Z 714.107,A -85,B 0,C 180,E1 -10282.493,E2 -10282.493} C_VEL
LIN {X 0,Y 572.865,Z 638.975,A -85,B 0,C 180,E1 -10283.536,E2 -10283.536} C_VEL
LIN {X 0,Y 570.434,Z 622.812,A -85,B 0,C 180,E1 -10283.838,E2 -10283.838} C_VEL
LIN {X 0,Y 571.063,Z 605.447,A -85,B 0,C 180,E1 -10286.989,E2 -10286.989} C_VEL
LIN {X 0,Y 571.402,Z 593.635,A -85,B 0,C 180,E1 -10289.161,E2 -10289.161} C_VEL
LIN {X 0,Y 570.428,Z 586.364,A -85,B 0,C 180,E1 -10290.562,E2 -10290.562} C_VEL
LIN {X 0,Y 570.309,Z 586.375,A -85,B 0,C 180,E1 -10293.551,E2 -10293.551} C_VEL
LIN {X 0,Y 570.346,Z 586.375,A -85,B 0,C 180,E1 -10296.12,E2 -10296.12} C_VEL
LIN {X 0,Y 570.263,Z 586.379,A -85,B 0,C 180,E1 -10299.302,E2 -10299.302} C_VEL
LIN {X 0,Y 570.303,Z 586.376,A -85,B 0,C 180,E1 -10301.546,E2 -10301.546} C_VEL
LIN {X 0,Y 570.309,Z 586.373,A -85,B 0,C 180,E1 -10304.574,E2 -10304.574} C_VEL
LIN {X 0,Y 570.307,Z 586.375,A -85,B 0,C 180,E1 -10307.506,E2 -10307.506} C_VEL
LIN {X 0,Y 570.288,Z 586.379,A -85,B 0,C 180,E1 -10310.306,E2 -10310.306} C_VEL
LIN {X 0,Y 570.314,Z 586.371,A -85,B 0,C 180,E1 -10313.001,E2 -10313.001} C_VEL
LIN {X 0,Y 570.315,Z 586.375,A -85,B 0,C 180,E1 -10315.6,E2 -10315.6} C_VEL
LIN {X 0,Y 570.325,Z 586.377,A -85,B 0,C 180,E1 -10318.122,E2 -10318.122} C_VEL
LIN {X 0,Y 570.312,Z 586.372,A -85,B 0,C 180,E1 -10320.692,E2 -10320.692} C_VEL
LIN {X 0,Y 570.3,Z 586.373,A -85,B 0,C 180,E1 -10322.971,E2 -10322.971} C_VEL
LIN {X 0,Y 570.33,Z 586.377,A -85,B 0,C 180,E1 -10326.091,E2 -10326.091} C_VEL
LIN {X 0,Y 570.318,Z 586.371,A -85,B 0,C 180,E1 -10327.088,E2 -10327.088} C_VEL
LIN {X 0,Y 569.651,Z 586.461,A -85,B 0,C 180,E1 -10327.678,E2 -10327.678} C_VEL
LIN {X 0,Y 566.782,Z 586.813,A -85,B 0,C 180,E1 -10328.634,E2 -10328.634} C_VEL
LIN {X 0,Y 564.364,Z 587.114,A -85,B 0,C 180,E1 -10329.404,E2 -10329.404} C_VEL
LIN {X 0,Y 563.339,Z 587.25,A -85,B 0,C 180,E1 -10329.998,E2 -10329.998} C_VEL
LIN {X 0,Y 563.263,Z 587.252,A -85,B 0,C 180,E1 -10330.199,E2 -10330.199} C_VEL
LIN {X 0,Y 563.33,Z 587.242,A -85,B 0,C 180,E1 -10333.217,E2 -10333.217} C_VEL
LIN {X 0,Y 563.369,Z 587.245,A -85,B 0,C 180,E1 -10335.877,E2 -10335.877} C_VEL
LIN {X 0,Y 563.379,Z 587.235,A -85,B 0,C 180,E1 -10339.17,E2 -10339.17} C_VEL
LIN {X 0,Y 563.384,Z 587.241,A -85,B 0,C 180,E1 -10342.139,E2 -10342.139} C_VEL
LIN {X 0,Y 563.475,Z 587.223,A -85,B 0,C 180,E1 -10345.008,E2 -10345.008} C_VEL
LIN {X 0,Y 563.469,Z 587.225,A -85,B 0,C 180,E1 -10348.575,E2 -10348.575} C_VEL
LIN {X 0,Y 563.594,Z 587.209,A -85,B 0,C 180,E1 -10350.712,E2 -10350.712} C_VEL
LIN {X 0,Y 563.455,Z 587.23,A -85,B 0,C 180,E1 -10354.277,E2 -10354.277} C_VEL
LIN {X 0,Y 563.414,Z 587.234,A -85,B 0,C 180,E1 -10356.424,E2 -10356.424} C_VEL
LIN {X 0,Y 563.342,Z 587.241,A -85,B 0,C 180,E1 -10358.581,E2 -10358.581} C_VEL
LIN {X 0,Y 563.329,Z 587.244,A -85,B 0,C 180,E1 -10361.475,E2 -10361.475} C_VEL
LIN {X 0,Y 563.354,Z 587.241,A -85,B 0,C 180,E1 -10364.399,E2 -10364.399} C_VEL
LIN {X 0,Y 563.296,Z 587.247,A -85,B 0,C 180,E1 -10367.363,E2 -10367.363} C_VEL
LIN {X 0,Y 563.28,Z 587.252,A -85,B 0,C 180,E1 -10369.618,E2 -10369.618} C_VEL
LIN {X 0,Y 563.298,Z 587.254,A -85,B 0,C 180,E1 -10371.903,E2 -10371.903} C_VEL
LIN {X 0,Y 563.258,Z 587.25,A -85,B 0,C 180,E1 -10374.799,E2 -10374.799} C_VEL
LIN {X 0,Y 563.287,Z 587.256,A -85,B 0,C 180,E1 -10378.009,E2 -10378.009} C_VEL
LIN {X 0,Y 563.284,Z 587.247,A -85,B 0,C 180,E1 -10380.907,E2 -10380.907} C_VEL
LIN {X 0,Y 563.274,Z 587.257,A -85,B 0,C 180,E1 -10384.027,E2 -10384.027} C_VEL
LIN {X 0,Y 563.304,Z 587.245,A -85,B 0,C 180,E1 -10386.645,E2 -10386.645} C_VEL
LIN {X 0,Y 563.259,Z 587.254,A -85,B 0,C 180,E1 -10389.557,E2 -10389.557} C_VEL
LIN {X 0,Y 563.266,Z 587.255,A -85,B 0,C 180,E1 -10392.184,E2 -10392.184} C_VEL
LIN {X 0,Y 563.268,Z 587.249,A -85,B 0,C 180,E1 -10395.139,E2 -10395.139} C_VEL
LIN {X 0,Y 563.267,Z 587.256,A -85,B 0,C 180,E1 -10397.817,E2 -10397.817} C_VEL
LIN {X 0,Y 563.221,Z 587.256,A -85,B 0,C 180,E1 -10400.636,E2 -10400.636} C_VEL
LIN {X 0,Y 563.293,Z 587.247,A -85,B 0,C 180,E1 -10403.354,E2 -10403.354} C_VEL
LIN {X 0,Y 563.26,Z 587.26,A -85,B 0,C 180,E1 -10405.972,E2 -10405.972} C_VEL
LIN {X 0,Y 563.286,Z 587.249,A -85,B 0,C 180,E1 -10408.516,E2 -10408.516} C_VEL
LIN {X 0,Y 563.262,Z 587.25,A -85,B 0,C 180,E1 -10410.989,E2 -10410.989} C_VEL
LIN {X 0,Y 563.243,Z 587.256,A -85,B 0,C 180,E1 -10413.558,E2 -10413.558} C_VEL
LIN {X 0,Y 563.276,Z 587.25,A -85,B 0,C 180,E1 -10416.552,E2 -10416.552} C_VEL
LIN {X 0,Y 563.318,Z 587.243,A -85,B 0,C 180,E1 -10418.864,E2 -10418.864} C_VEL
LIN {X 0,Y 563.288,Z 587.255,A -85,B 0,C 180,E1 -10421.888,E2 -10421.888} C_VEL
LIN {X 0,Y 563.331,Z 587.241,A -85,B 0,C 180,E1 -10424.864,E2 -10424.864} C_VEL
LIN {X 0,Y 563.297,Z 587.245,A -85,B 0,C 180,E1 -10427.067,E2 -10427.067} C_VEL
LIN {X 0,Y 563.353,Z 587.248,A -85,B 0,C 180,E1 -10429.976,E2 -10429.976} C_VEL
LIN {X 0,Y 563.402,Z 587.232,A -85,B 0,C 180,E1 -10432.859,E2 -10432.859} C_VEL
LIN {X 0,Y 563.458,Z 587.225,A -85,B 0,C 180,E1 -10435.008,E2 -10435.008} C_VEL
LIN {X 0,Y 563.478,Z 587.224,A -85,B 0,C 180,E1 -10438.576,E2 -10438.576} C_VEL
LIN {X 0,Y 563.596,Z 587.209,A -85,B 0,C 180,E1 -10440.712,E2 -10440.712} C_VEL
LIN {X 0,Y 563.438,Z 587.232,A -85,B 0,C 180,E1 -10444.278,E2 -10444.278} C_VEL
LIN {X 0,Y 563.42,Z 587.233,A -85,B 0,C 180,E1 -10446.424,E2 -10446.424} C_VEL
LIN {X 0,Y 563.313,Z 587.245,A -85,B 0,C 180,E1 -10449.303,E2 -10449.303} C_VEL
LIN {X 0,Y 563.328,Z 587.244,A -85,B 0,C 180,E1 -10451.475,E2 -10451.475} C_VEL
LIN {X 0,Y 563.33,Z 587.244,A -85,B 0,C 180,E1 -10454.4,E2 -10454.4} C_VEL
LIN {X 0,Y 563.263,Z 587.251,A -85,B 0,C 180,E1 -10457.365,E2 -10457.365} C_VEL
LIN {X 0,Y 563.258,Z 587.255,A -85,B 0,C 180,E1 -10459.619,E2 -10459.619} C_VEL
LIN {X 0,Y 563.281,Z 587.256,A -85,B 0,C 180,E1 -10461.904,E2 -10461.904} C_VEL
LIN {X 0,Y 563.265,Z 587.249,A -85,B 0,C 180,E1 -10465.012,E2 -10465.012} C_VEL
LIN {X 0,Y 563.28,Z 587.253,A -85,B 0,C 180,E1 -10468.199,E2 -10468.199} C_VEL
LIN {X 0,Y 563.229,Z 587.254,A -85,B 0,C 180,E1 -10470.896,E2 -10470.896} C_VEL
LIN {X 0,Y 563.224,Z 587.258,A -85,B 0,C 180,E1 -10473.568,E2 -10473.568} C_VEL
LIN {X 0,Y 563.272,Z 587.256,A -85,B 0,C 180,E1 -10476.071,E2 -10476.071} C_VEL
LIN {X 0,Y 563.208,Z 587.259,A -85,B 0,C 180,E1 -10478.45,E2 -10478.45} C_VEL
LIN {X 0,Y 563.229,Z 587.255,A -85,B 0,C 180,E1 -10481.233,E2 -10481.233} C_VEL
LIN {X 0,Y 563.248,Z 587.258,A -85,B 0,C 180,E1 -10484.139,E2 -10484.139} C_VEL
LIN {X 0,Y 563.255,Z 587.251,A -85,B 0,C 180,E1 -10487.198,E2 -10487.198} C_VEL
LIN {X 0,Y 563.234,Z 587.259,A -85,B 0,C 180,E1 -10489.709,E2 -10489.709} C_VEL
LIN {X 0,Y 563.207,Z 587.257,A -85,B 0,C 180,E1 -10492.745,E2 -10492.745} C_VEL
LIN {X 0,Y 563.254,Z 587.251,A -85,B 0,C 180,E1 -10495.16,E2 -10495.16} C_VEL
LIN {X 0,Y 563.247,Z 587.258,A -85,B 0,C 180,E1 -10497.74,E2 -10497.74} C_VEL
LIN {X 0,Y 563.246,Z 587.254,A -85,B 0,C 180,E1 -10500.518,E2 -10500.518} C_VEL
LIN {X 0,Y 563.241,Z 587.254,A -85,B 0,C 180,E1 -10503.404,E2 -10503.404} C_VEL
LIN {X 0,Y 563.307,Z 587.426,A -85,B 0,C 180,E1 -10506.31,E2 -10506.31} C_VEL
LIN {X 0,Y 565.348,Z 599.064,A -85,B 0,C 180,E1 -10508.313,E2 -10508.313} C_VEL
LIN {X 0,Y 564.607,Z 615.697,A -85,B 0,C 180,E1 -10511.006,E2 -10511.006} C_VEL
LIN {X 0,Y 563.795,Z 634.134,A -85,B 0,C 180,E1 -10513.953,E2 -10513.953} C_VEL
LIN {X 0,Y 563.289,Z 647.346,A -85,B 0,C 180,E1 -10516.046,E2 -10516.046} C_VEL
LIN {X 0,Y 565.827,Z 667.574,A -85,B 0,C 180,E1 -10516.397,E2 -10516.397} C_VEL
LIN {X 0,Y 564.951,Z 753.778,A -85,B 0,C 180,E1 -10517.628,E2 -10517.628} C_VEL
LIN {X 0,Y 564.774,Z 763.929,A -85,B 0,C 180,E1 -10517.851,E2 -10517.851} C_VEL
LIN {X 0,Y 564.532,Z 773.474,A -85,B 0,C 180,E1 -10518.141,E2 -10518.141} C_VEL
LIN {X 0,Y 564.261,Z 783.589,A -85,B 0,C 180,E1 -10518.544,E2 -10518.544} C_VEL
LIN {X 0,Y 564.016,Z 793.966,A -85,B 0,C 180,E1 -10519.071,E2 -10519.071} C_VEL
LIN {X 0,Y 563.58,Z 804.087,A -85,B 0,C 180,E1 -10519.708,E2 -10519.708} C_VEL
LIN {X 0,Y 563.297,Z 812.39,A -85,B 0,C 180,E1 -10520.336,E2 -10520.336} C_VEL
LIN {X 0,Y 562.93,Z 820.39,A -85,B 0,C 180,E1 -10521.052,E2 -10521.052} C_VEL
LIN {X 0,Y 562.637,Z 828.686,A -85,B 0,C 180,E1 -10521.949,E2 -10521.949} C_VEL
LIN {X 0,Y 562.391,Z 835.591,A -85,B 0,C 180,E1 -10522.845,E2 -10522.845} C_VEL
LIN {X 0,Y 562.241,Z 840.342,A -85,B 0,C 180,E1 -10523.562,E2 -10523.562} C_VEL
LIN {X 0,Y 562.101,Z 846.162,A -85,B 0,C 180,E1 -10524.638,E2 -10524.638} C_VEL
LIN {X 0,Y 562.016,Z 850.728,A -85,B 0,C 180,E1 -10525.712,E2 -10525.712} C_VEL
LIN {X 0,Y 561.983,Z 853.079,A -85,B 0,C 180,E1 -10526.427,E2 -10526.427} C_VEL
LIN {X 0,Y 561.919,Z 856.617,A -85,B 0,C 180,E1 -10527.857,E2 -10527.857} C_VEL
LIN {X 0,Y 561.904,Z 858.279,A -85,B 0,C 180,E1 -10529.286,E2 -10529.286} C_VEL
LIN {X 0,Y 561.894,Z 858.592,A -85,B 0,C 180,E1 -10530,E2 -10530} C_VEL
LIN {X 0,Y 561.884,Z 857.8,A -85,B 0,C 180,E1 -10531.429,E2 -10531.429} C_VEL
LIN {X 0,Y 561.92,Z 856.796,A -85,B 0,C 180,E1 -10532.143,E2 -10532.143} C_VEL
LIN {X 0,Y 561.983,Z 853.538,A -85,B 0,C 180,E1 -10533.573,E2 -10533.573} C_VEL
LIN {X 0,Y 562.02,Z 850.024,A -85,B 0,C 180,E1 -10534.611,E2 -10534.611} C_VEL
LIN {X 0,Y 562.176,Z 845.067,A -85,B 0,C 180,E1 -10535.721,E2 -10535.721} C_VEL
LIN {X 0,Y 562.35,Z 838.968,A -85,B 0,C 180,E1 -10536.796,E2 -10536.796} C_VEL
LIN {X 0,Y 562.567,Z 832.798,A -85,B 0,C 180,E1 -10537.692,E2 -10537.692} C_VEL
LIN {X 0,Y 562.818,Z 825.361,A -85,B 0,C 180,E1 -10538.589,E2 -10538.589} C_VEL
LIN {X 0,Y 563.298,Z 816.329,A -85,B 0,C 180,E1 -10539.483,E2 -10539.483} C_VEL
LIN {X 0,Y 563.695,Z 807.656,A -85,B 0,C 180,E1 -10540.199,E2 -10540.199} C_VEL
LIN {X 0,Y 564.064,Z 798.317,A -85,B 0,C 180,E1 -10540.841,E2 -10540.841} C_VEL
LIN {X 0,Y 564.36,Z 789.013,A -85,B 0,C 180,E1 -10541.372,E2 -10541.372} C_VEL
LIN {X 0,Y 564.702,Z 778.43,A -85,B 0,C 180,E1 -10541.855,E2 -10541.855} C_VEL
LIN {X 0,Y 564.951,Z 767.651,A -85,B 0,C 180,E1 -10542.236,E2 -10542.236} C_VEL
LIN {X 0,Y 565.325,Z 756.139,A -85,B 0,C 180,E1 -10542.523,E2 -10542.523} C_VEL
LIN {X 0,Y 565.578,Z 736.305,A -85,B 0,C 180,E1 -10542.835,E2 -10542.835} C_VEL
LIN {X 0,Y 566.283,Z 666.546,A -85,B 0,C 180,E1 -10543.863,E2 -10543.863} C_VEL
LIN {X 0,Y 564.273,Z 651.572,A -85,B 0,C 180,E1 -10544.155,E2 -10544.155} C_VEL
LIN {X 0,Y 563.494,Z 646.478,A -85,B 0,C 180,E1 -10544.268,E2 -10544.268} C_VEL
LIN {X 0,Y 564.325,Z 627.542,A -85,B 0,C 180,E1 -10547.331,E2 -10547.331} C_VEL
LIN {X 0,Y 565.283,Z 609.634,A -85,B 0,C 180,E1 -10550.301,E2 -10550.301} C_VEL
LIN {X 0,Y 565.691,Z 600.756,A -85,B 0,C 180,E1 -10551.806,E2 -10551.806} C_VEL
LIN {X 0,Y 564.016,Z 590.961,A -85,B 0,C 180,E1 -10553.61,E2 -10553.61} C_VEL
LIN {X 0,Y 563.295,Z 587.255,A -85,B 0,C 180,E1 -10554.354,E2 -10554.354} C_VEL
LIN {X 0,Y 563.251,Z 587.262,A -85,B 0,C 180,E1 -10557.395,E2 -10557.395} C_VEL
LIN {X 0,Y 563.231,Z 587.265,A -85,B 0,C 180,E1 -10559.831,E2 -10559.831} C_VEL
LIN {X 0,Y 563.241,Z 587.258,A -85,B 0,C 180,E1 -10562.327,E2 -10562.327} C_VEL
LIN {X 0,Y 563.272,Z 587.251,A -85,B 0,C 180,E1 -10564.892,E2 -10564.892} C_VEL
LIN {X 0,Y 563.248,Z 587.256,A -85,B 0,C 180,E1 -10567.543,E2 -10567.543} C_VEL
LIN {X 0,Y 563.247,Z 587.25,A -85,B 0,C 180,E1 -10570.66,E2 -10570.66} C_VEL
LIN {X 0,Y 563.258,Z 587.256,A -85,B 0,C 180,E1 -10573.154,E2 -10573.154} C_VEL
LIN {X 0,Y 563.252,Z 587.256,A -85,B 0,C 180,E1 -10575.861,E2 -10575.861} C_VEL
LIN {X 0,Y 563.25,Z 587.255,A -85,B 0,C 180,E1 -10578.258,E2 -10578.258} C_VEL
LIN {X 0,Y 563.223,Z 587.26,A -85,B 0,C 180,E1 -10580.635,E2 -10580.635} C_VEL
LIN {X 0,Y 563.328,Z 587.244,A -85,B 0,C 180,E1 -10583.922,E2 -10583.922} C_VEL
LIN {X 0,Y 563.259,Z 587.258,A -85,B 0,C 180,E1 -10586.827,E2 -10586.827} C_VEL
LIN {X 0,Y 563.273,Z 587.252,A -85,B 0,C 180,E1 -10589.346,E2 -10589.346} C_VEL
LIN {X 0,Y 563.293,Z 587.249,A -85,B 0,C 180,E1 -10591.991,E2 -10591.991} C_VEL
LIN {X 0,Y 563.266,Z 587.255,A -85,B 0,C 180,E1 -10595.202,E2 -10595.202} C_VEL
LIN {X 0,Y 563.301,Z 587.253,A -85,B 0,C 180,E1 -10598.097,E2 -10598.097} C_VEL
LIN {X 0,Y 563.301,Z 587.254,A -85,B 0,C 180,E1 -10601.137,E2 -10601.137} C_VEL
LIN {X 0,Y 563.287,Z 587.257,A -85,B 0,C 180,E1 -10604.123,E2 -10604.123} C_VEL
LIN {X 0,Y 563.358,Z 587.248,A -85,B 0,C 180,E1 -10606.335,E2 -10606.335} C_VEL
LIN {X 0,Y 563.367,Z 587.441,A -85,B 0,C 180,E1 -10608.569,E2 -10608.569} C_VEL
LIN {X 0,Y 564.888,Z 595.895,A -85,B 0,C 180,E1 -10610.363,E2 -10610.363} C_VEL
LIN {X 0,Y 564.936,Z 603.134,A -85,B 0,C 180,E1 -10611.802,E2 -10611.802} C_VEL
LIN {X 0,Y 564.055,Z 617.987,A -85,B 0,C 180,E1 -10614.656,E2 -10614.656} C_VEL
LIN {X 0,Y 563.701,Z 624.003,A -85,B 0,C 180,E1 -10615.791,E2 -10615.791} C_VEL
LIN {X 0,Y 566.562,Z 640.27,A -85,B 0,C 180,E1 -10616.145,E2 -10616.145} C_VEL
LIN {X 0,Y 565.566,Z 709.096,A -85,B 0,C 180,E1 -10617.16,E2 -10617.16} C_VEL
LIN {X 0,Y 565.207,Z 731.735,A -85,B 0,C 180,E1 -10617.514,E2 -10617.514} C_VEL
LIN {X 0,Y 565.004,Z 743.196,A -85,B 0,C 180,E1 -10617.802,E2 -10617.802} C_VEL
LIN {X 0,Y 564.716,Z 756.217,A -85,B 0,C 180,E1 -10618.267,E2 -10618.267} C_VEL
LIN {X 0,Y 564.466,Z 767.94,A -85,B 0,C 180,E1 -10618.844,E2 -10618.844} C_VEL
LIN {X 0,Y 564.092,Z 779.203,A -85,B 0,C 180,E1 -10619.555,E2 -10619.555} C_VEL
LIN {X 0,Y 563.733,Z 788.425,A -85,B 0,C 180,E1 -10620.267,E2 -10620.267} C_VEL
LIN {X 0,Y 563.372,Z 795.359,A -85,B 0,C 180,E1 -10620.89,E2 -10620.89} C_VEL
LIN {X 0,Y 562.914,Z 803.604,A -85,B 0,C 180,E1 -10621.782,E2 -10621.782} C_VEL
LIN {X 0,Y 562.667,Z 810.459,A -85,B 0,C 180,E1 -10622.675,E2 -10622.675} C_VEL
LIN {X 0,Y 562.337,Z 816.218,A -85,B 0,C 180,E1 -10623.57,E2 -10623.57} C_VEL
LIN {X 0,Y 562.234,Z 821.929,A -85,B 0,C 180,E1 -10624.682,E2 -10624.682} C_VEL
LIN {X 0,Y 562.104,Z 826.429,A -85,B 0,C 180,E1 -10625.809,E2 -10625.809} C_VEL
LIN {X 0,Y 562.05,Z 828.481,A -85,B 0,C 180,E1 -10626.44,E2 -10626.44} C_VEL
LIN {X 0,Y 561.843,Z 831.734,A -85,B 0,C 180,E1 -10627.882,E2 -10627.882} C_VEL
LIN {X 0,Y 561.865,Z 832.706,A -85,B 0,C 180,E1 -10628.603,E2 -10628.603} C_VEL
LIN {X 0,Y 561.897,Z 833.442,A -85,B 0,C 180,E1 -10630.05,E2 -10630.05} C_VEL
LIN {X 0,Y 561.837,Z 832.361,A -85,B 0,C 180,E1 -10631.506,E2 -10631.506} C_VEL
LIN {X 0,Y 561.857,Z 831.305,A -85,B 0,C 180,E1 -10632.235,E2 -10632.235} C_VEL
LIN {X 0,Y 562.007,Z 827.554,A -85,B 0,C 180,E1 -10633.698,E2 -10633.698} C_VEL
LIN {X 0,Y 562.064,Z 825.088,A -85,B 0,C 180,E1 -10634.432,E2 -10634.432} C_VEL
LIN {X 0,Y 562.26,Z 819.225,A -85,B 0,C 180,E1 -10635.721,E2 -10635.721} C_VEL
LIN {X 0,Y 562.386,Z 813.962,A -85,B 0,C 180,E1 -10636.646,E2 -10636.646} C_VEL
LIN {X 0,Y 562.595,Z 807.562,A -85,B 0,C 180,E1 -10637.573,E2 -10637.573} C_VEL
LIN {X 0,Y 562.92,Z 799.785,A -85,B 0,C 180,E1 -10638.499,E2 -10638.499} C_VEL
LIN {X 0,Y 563.268,Z 791.272,A -85,B 0,C 180,E1 -10639.339,E2 -10639.339} C_VEL
LIN {X 0,Y 563.516,Z 783.516,A -85,B 0,C 180,E1 -10639.988,E2 -10639.988} C_VEL
LIN {X 0,Y 563.871,Z 774.169,A -85,B 0,C 180,E1 -10640.638,E2 -10640.638} C_VEL
LIN {X 0,Y 564.204,Z 764.49,A -85,B 0,C 180,E1 -10641.193,E2 -10641.193} C_VEL
LIN {X 0,Y 564.507,Z 753.201,A -85,B 0,C 180,E1 -10641.705,E2 -10641.705} C_VEL
LIN {X 0,Y 564.673,Z 742.181,A -85,B 0,C 180,E1 -10642.086,E2 -10642.086} C_VEL
LIN {X 0,Y 564.914,Z 732.101,A -85,B 0,C 180,E1 -10642.34,E2 -10642.34} C_VEL
LIN {X 0,Y 565.219,Z 712.913,A -85,B 0,C 180,E1 -10642.64,E2 -10642.64} C_VEL
LIN {X 0,Y 565.832,Z 638.995,A -85,B 0,C 180,E1 -10643.686,E2 -10643.686} C_VEL
LIN {X 0,Y 563.419,Z 622.955,A -85,B 0,C 180,E1 -10643.989,E2 -10643.989} C_VEL
LIN {X 0,Y 564.061,Z 605.721,A -85,B 0,C 180,E1 -10647.152,E2 -10647.152} C_VEL
LIN {X 0,Y 564.39,Z 594.231,A -85,B 0,C 180,E1 -10649.288,E2 -10649.288} C_VEL
LIN {X 0,Y 563.361,Z 587.244,A -85,B 0,C 180,E1 -10650.648,E2 -10650.648} C_VEL
LIN {X 0,Y 563.266,Z 587.258,A -85,B 0,C 180,E1 -10654.027,E2 -10654.027} C_VEL
LIN {X 0,Y 563.274,Z 587.249,A -85,B 0,C 180,E1 -10656.647,E2 -10656.647} C_VEL
LIN {X 0,Y 563.26,Z 587.253,A -85,B 0,C 180,E1 -10659.556,E2 -10659.556} C_VEL
LIN {X 0,Y 563.269,Z 587.255,A -85,B 0,C 180,E1 -10662.183,E2 -10662.183} C_VEL
LIN {X 0,Y 563.27,Z 587.249,A -85,B 0,C 180,E1 -10665.138,E2 -10665.138} C_VEL
LIN {X 0,Y 563.268,Z 587.256,A -85,B 0,C 180,E1 -10667.816,E2 -10667.816} C_VEL
LIN {X 0,Y 563.219,Z 587.256,A -85,B 0,C 180,E1 -10670.635,E2 -10670.635} C_VEL
LIN {X 0,Y 563.322,Z 587.251,A -85,B 0,C 180,E1 -10673.922,E2 -10673.922} C_VEL
LIN {X 0,Y 563.249,Z 587.251,A -85,B 0,C 180,E1 -10676.826,E2 -10676.826} C_VEL
LIN {X 0,Y 563.273,Z 587.25,A -85,B 0,C 180,E1 -10679.346,E2 -10679.346} C_VEL
LIN {X 0,Y 563.287,Z 587.256,A -85,B 0,C 180,E1 -10681.991,E2 -10681.991} C_VEL
LIN {X 0,Y 563.26,Z 587.251,A -85,B 0,C 180,E1 -10685.201,E2 -10685.201} C_VEL
LIN {X 0,Y 563.294,Z 587.253,A -85,B 0,C 180,E1 -10688.096,E2 -10688.096} C_VEL
LIN {X 0,Y 563.263,Z 587.252,A -85,B 0,C 180,E1 -10690.199,E2 -10690.199} C_VEL
LIN {X 0,Y 562.629,Z 587.333,A -85,B 0,C 180,E1 -10690.796,E2 -10690.796} C_VEL
LIN {X 0,Y 559.826,Z 587.684,A -85,B 0,C 180,E1 -10691.765,E2 -10691.765} C_VEL
LIN {X 0,Y 557.429,Z 587.978,A -85,B 0,C 180,E1 -10692.545,E2 -10692.545} C_VEL
LIN {X 0,Y 556.377,Z 588.108,A -85,B 0,C 180,E1 -10693.146,E2 -10693.146} C_VEL
LIN {X 0,Y 556.279,Z 588.121,A -85,B 0,C 180,E1 -10693.35,E2 -10693.35} C_VEL
LIN {X 0,Y 556.326,Z 588.12,A -85,B 0,C 180,E1 -10696.159,E2 -10696.159} C_VEL
LIN {X 0,Y 556.352,Z 588.111,A -85,B 0,C 180,E1 -10699.114,E2 -10699.114} C_VEL
LIN {X 0,Y 556.335,Z 588.121,A -85,B 0,C 180,E1 -10702.039,E2 -10702.039} C_VEL
LIN {X 0,Y 556.435,Z 588.1,A -85,B 0,C 180,E1 -10704.945,E2 -10704.945} C_VEL
LIN {X 0,Y 556.417,Z 588.104,A -85,B 0,C 180,E1 -10708.557,E2 -10708.557} C_VEL
LIN {X 0,Y 556.545,Z 588.087,A -85,B 0,C 180,E1 -10710.721,E2 -10710.721} C_VEL
LIN {X 0,Y 556.416,Z 588.106,A -85,B 0,C 180,E1 -10714.332,E2 -10714.332} C_VEL
LIN {X 0,Y 556.374,Z 588.11,A -85,B 0,C 180,E1 -10716.506,E2 -10716.506} C_VEL
LIN {X 0,Y 556.259,Z 588.124,A -85,B 0,C 180,E1 -10719.421,E2 -10719.421} C_VEL
LIN {X 0,Y 556.281,Z 588.124,A -85,B 0,C 180,E1 -10721.623,E2 -10721.623} C_VEL
LIN {X 0,Y 556.322,Z 588.116,A -85,B 0,C 180,E1 -10724.585,E2 -10724.585} C_VEL
LIN {X 0,Y 556.246,Z 588.127,A -85,B 0,C 180,E1 -10727.591,E2 -10727.591} C_VEL
LIN {X 0,Y 556.242,Z 588.132,A -85,B 0,C 180,E1 -10729.877,E2 -10729.877} C_VEL
LIN {X 0,Y 556.239,Z 588.13,A -85,B 0,C 180,E1 -10732.196,E2 -10732.196} C_VEL
LIN {X 0,Y 556.222,Z 588.127,A -85,B 0,C 180,E1 -10734.95,E2 -10734.95} C_VEL
LIN {X 0,Y 556.247,Z 588.13,A -85,B 0,C 180,E1 -10738.182,E2 -10738.182} C_VEL
LIN {X 0,Y 556.242,Z 588.124,A -85,B 0,C 180,E1 -10741.099,E2 -10741.099} C_VEL
LIN {X 0,Y 556.242,Z 588.131,A -85,B 0,C 180,E1 -10743.789,E2 -10743.789} C_VEL
LIN {X 0,Y 556.281,Z 588.124,A -85,B 0,C 180,E1 -10746.308,E2 -10746.308} C_VEL
LIN {X 0,Y 556.2,Z 588.129,A -85,B 0,C 180,E1 -10749.026,E2 -10749.026} C_VEL
LIN {X 0,Y 556.203,Z 588.137,A -85,B 0,C 180,E1 -10751.87,E2 -10751.87} C_VEL
LIN {X 0,Y 556.246,Z 588.124,A -85,B 0,C 180,E1 -10754.843,E2 -10754.843} C_VEL
LIN {X 0,Y 556.21,Z 588.138,A -85,B 0,C 180,E1 -10757.987,E2 -10757.987} C_VEL
LIN {X 0,Y 556.231,Z 588.131,A -85,B 0,C 180,E1 -10760.188,E2 -10760.188} C_VEL
LIN {X 0,Y 556.256,Z 588.123,A -85,B 0,C 180,E1 -10762.813,E2 -10762.813} C_VEL
LIN {X 0,Y 556.237,Z 588.127,A -85,B 0,C 180,E1 -10765.483,E2 -10765.483} C_VEL
LIN {X 0,Y 556.222,Z 588.135,A -85,B 0,C 180,E1 -10768.069,E2 -10768.069} C_VEL
LIN {X 0,Y 556.237,Z 588.126,A -85,B 0,C 180,E1 -10770.587,E2 -10770.587} C_VEL
LIN {X 0,Y 556.221,Z 588.129,A -85,B 0,C 180,E1 -10773.392,E2 -10773.392} C_VEL
LIN {X 0,Y 556.229,Z 588.131,A -85,B 0,C 180,E1 -10776.237,E2 -10776.237} C_VEL
LIN {X 0,Y 556.256,Z 588.123,A -85,B 0,C 180,E1 -10778.72,E2 -10778.72} C_VEL
LIN {X 0,Y 556.235,Z 588.13,A -85,B 0,C 180,E1 -10781.651,E2 -10781.651} C_VEL
LIN {X 0,Y 556.231,Z 588.135,A -85,B 0,C 180,E1 -10783.917,E2 -10783.917} C_VEL
LIN {X 0,Y 556.322,Z 588.121,A -85,B 0,C 180,E1 -10786.16,E2 -10786.16} C_VEL
LIN {X 0,Y 556.356,Z 588.11,A -85,B 0,C 180,E1 -10789.115,E2 -10789.115} C_VEL
LIN {X 0,Y 556.34,Z 588.121,A -85,B 0,C 180,E1 -10792.04,E2 -10792.04} C_VEL
LIN {X 0,Y 556.375,Z 588.113,A -85,B 0,C 180,E1 -10794.22,E2 -10794.22} C_VEL
LIN {X 0,Y 556.345,Z 588.115,A -85,B 0,C 180,E1 -10796.391,E2 -10796.391} C_VEL
LIN {X 0,Y 556.593,Z 588.09,A -85,B 0,C 180,E1 -10800,E2 -10800} C_VEL
LIN {X 0,Y 556.344,Z 588.116,A -85,B 0,C 180,E1 -10803.609,E2 -10803.609} C_VEL
LIN {X 0,Y 556.449,Z 588.107,A -85,B 0,C 180,E1 -10806.049,E2 -10806.049} C_VEL
LIN {X 0,Y 556.31,Z 588.116,A -85,B 0,C 180,E1 -10808.69,E2 -10808.69} C_VEL
LIN {X 0,Y 556.357,Z 588.11,A -85,B 0,C 180,E1 -10810.886,E2 -10810.886} C_VEL
LIN {X 0,Y 556.318,Z 588.121,A -85,B 0,C 180,E1 -10814.191,E2 -10814.191} C_VEL
LIN {X 0,Y 556.227,Z 588.126,A -85,B 0,C 180,E1 -10816.853,E2 -10816.853} C_VEL
LIN {X 0,Y 556.219,Z 588.135,A -85,B 0,C 180,E1 -10819.878,E2 -10819.878} C_VEL
LIN {X 0,Y 556.227,Z 588.132,A -85,B 0,C 180,E1 -10822.197,E2 -10822.197} C_VEL
LIN {X 0,Y 556.225,Z 588.126,A -85,B 0,C 180,E1 -10824.949,E2 -10824.949} C_VEL
LIN {X 0,Y 556.23,Z 588.132,A -85,B 0,C 180,E1 -10827.771,E2 -10827.771} C_VEL
LIN {X 0,Y 556.198,Z 588.135,A -85,B 0,C 180,E1 -10830.248,E2 -10830.248} C_VEL
LIN {X 0,Y 556.178,Z 588.132,A -85,B 0,C 180,E1 -10832.788,E2 -10832.788} C_VEL
LIN {X 0,Y 556.197,Z 588.132,A -85,B 0,C 180,E1 -10835.401,E2 -10835.401} C_VEL
LIN {X 0,Y 556.178,Z 588.139,A -85,B 0,C 180,E1 -10838.105,E2 -10838.105} C_VEL
LIN {X 0,Y 556.194,Z 588.13,A -85,B 0,C 180,E1 -10840.921,E2 -10840.921} C_VEL
LIN {X 0,Y 556.212,Z 588.136,A -85,B 0,C 180,E1 -10843.838,E2 -10843.838} C_VEL
LIN {X 0,Y 556.212,Z 588.134,A -85,B 0,C 180,E1 -10846.162,E2 -10846.162} C_VEL
LIN {X 0,Y 556.203,Z 588.129,A -85,B 0,C 180,E1 -10849.092,E2 -10849.092} C_VEL
LIN {X 0,Y 556.17,Z 588.142,A -85,B 0,C 180,E1 -10851.895,E2 -10851.895} C_VEL
LIN {X 0,Y 556.196,Z 588.131,A -85,B 0,C 180,E1 -10854.599,E2 -10854.599} C_VEL
LIN {X 0,Y 556.19,Z 588.134,A -85,B 0,C 180,E1 -10857.541,E2 -10857.541} C_VEL
LIN {X 0,Y 556.217,Z 588.129,A -85,B 0,C 180,E1 -10860.585,E2 -10860.585} C_VEL
LIN {X 0,Y 556.215,Z 588.129,A -85,B 0,C 180,E1 -10863.394,E2 -10863.394} C_VEL
LIN {X 0,Y 556.257,Z 588.286,A -85,B 0,C 180,E1 -10866.188,E2 -10866.188} C_VEL
LIN {X 0,Y 558.309,Z 599.732,A -85,B 0,C 180,E1 -10868.185,E2 -10868.185} C_VEL
LIN {X 0,Y 557.759,Z 613.002,A -85,B 0,C 180,E1 -10870.367,E2 -10870.367} C_VEL
LIN {X 0,Y 556.842,Z 632.68,A -85,B 0,C 180,E1 -10873.559,E2 -10873.559} C_VEL
LIN {X 0,Y 556.272,Z 647.213,A -85,B 0,C 180,E1 -10875.894,E2 -10875.894} C_VEL
LIN {X 0,Y 558.852,Z 668.76,A -85,B 0,C 180,E1 -10876.27,E2 -10876.27} C_VEL
LIN {X 0,Y 557.956,Z 753.975,A -85,B 0,C 180,E1 -10877.517,E2 -10877.517} C_VEL
LIN {X 0,Y 557.749,Z 763.976,A -85,B 0,C 180,E1 -10877.742,E2 -10877.742} C_VEL
LIN {X 0,Y 557.506,Z 773.456,A -85,B 0,C 180,E1 -10878.036,E2 -10878.036} C_VEL
LIN {X 0,Y 557.213,Z 783.924,A -85,B 0,C 180,E1 -10878.462,E2 -10878.462} C_VEL
LIN {X 0,Y 556.959,Z 794.587,A -85,B 0,C 180,E1 -10879.019,E2 -10879.019} C_VEL
LIN {X 0,Y 556.575,Z 803.389,A -85,B 0,C 180,E1 -10879.577,E2 -10879.577} C_VEL
LIN {X 0,Y 556.234,Z 812.82,A -85,B 0,C 180,E1 -10880.304,E2 -10880.304} C_VEL
LIN {X 0,Y 555.812,Z 821.591,A -85,B 0,C 180,E1 -10881.119,E2 -10881.119} C_VEL
LIN {X 0,Y 555.582,Z 828.231,A -85,B 0,C 180,E1 -10881.846,E2 -10881.846} C_VEL
LIN {X 0,Y 555.311,Z 835.194,A -85,B 0,C 180,E1 -10882.754,E2 -10882.754} C_VEL
LIN {X 0,Y 555.127,Z 841.012,A -85,B 0,C 180,E1 -10883.661,E2 -10883.661} C_VEL
LIN {X 0,Y 555.012,Z 845.844,A -85,B 0,C 180,E1 -10884.569,E2 -10884.569} C_VEL
LIN {X 0,Y 554.909,Z 850.615,A -85,B 0,C 180,E1 -10885.704,E2 -10885.704} C_VEL
LIN {X 0,Y 554.885,Z 854.781,A -85,B 0,C 180,E1 -10887.106,E2 -10887.106} C_VEL
LIN {X 0,Y 554.845,Z 856.403,A -85,B 0,C 180,E1 -10887.83,E2 -10887.83} C_VEL
LIN {X 0,Y 554.815,Z 858.104,A -85,B 0,C 180,E1 -10889.277,E2 -10889.277} C_VEL
LIN {X 0,Y 554.804,Z 858.417,A -85,B 0,C 180,E1 -10890,E2 -10890} C_VEL
LIN {X 0,Y 554.801,Z 857.671,A -85,B 0,C 180,E1 -10891.447,E2 -10891.447} C_VEL
LIN {X 0,Y 554.845,Z 856.664,A -85,B 0,C 180,E1 -10892.171,E2 -10892.171} C_VEL
LIN {X 0,Y 554.889,Z 853.442,A -85,B 0,C 180,E1 -10893.619,E2 -10893.619} C_VEL
LIN {X 0,Y 554.945,Z 849.791,A -85,B 0,C 180,E1 -10894.706,E2 -10894.706} C_VEL
LIN {X 0,Y 555.096,Z 844.999,A -85,B 0,C 180,E1 -10895.794,E2 -10895.794} C_VEL
LIN {X 0,Y 555.298,Z 838.913,A -85,B 0,C 180,E1 -10896.883,E2 -10896.883} C_VEL
LIN {X 0,Y 555.517,Z 832.755,A -85,B 0,C 180,E1 -10897.79,E2 -10897.79} C_VEL
LIN {X 0,Y 555.784,Z 825.332,A -85,B 0,C 180,E1 -10898.699,E2 -10898.699} C_VEL
LIN {X 0,Y 556.297,Z 816.316,A -85,B 0,C 180,E1 -10899.604,E2 -10899.604} C_VEL
LIN {X 0,Y 556.71,Z 807.664,A -85,B 0,C 180,E1 -10900.329,E2 -10900.329} C_VEL
LIN {X 0,Y 557.078,Z 798.621,A -85,B 0,C 180,E1 -10900.963,E2 -10900.963} C_VEL
LIN {X 0,Y 557.432,Z 788.624,A -85,B 0,C 180,E1 -10901.54,E2 -10901.54} C_VEL
LIN {X 0,Y 557.804,Z 777.496,A -85,B 0,C 180,E1 -10902.05,E2 -10902.05} C_VEL
LIN {X 0,Y 558.076,Z 767.337,A -85,B 0,C 180,E1 -10902.412,E2 -10902.412} C_VEL
LIN {X 0,Y 558.441,Z 755.879,A -85,B 0,C 180,E1 -10902.703,E2 -10902.703} C_VEL
LIN {X 0,Y 558.746,Z 734.743,A -85,B 0,C 180,E1 -10903.041,E2 -10903.041} C_VEL
LIN {X 0,Y 559.478,Z 667.153,A -85,B 0,C 180,E1 -10904.059,E2 -10904.059} C_VEL
LIN {X 0,Y 556.916,Z 648.69,A -85,B 0,C 180,E1 -10904.432,E2 -10904.432} C_VEL
LIN {X 0,Y 556.526,Z 646.299,A -85,B 0,C 180,E1 -10904.492,E2 -10904.492} C_VEL
LIN {X 0,Y 557.387,Z 627.71,A -85,B 0,C 180,E1 -10907.554,E2 -10907.554} C_VEL
LIN {X 0,Y 558.515,Z 608.731,A -85,B 0,C 180,E1 -10910.75,E2 -10910.75} C_VEL
LIN {X 0,Y 558.705,Z 601.043,A -85,B 0,C 180,E1 -10912.093,E2 -10912.093} C_VEL
LIN {X 0,Y 556.251,Z 588.132,A -85,B 0,C 180,E1 -10914.554,E2 -10914.554} C_VEL
LIN {X 0,Y 556.206,Z 588.142,A -85,B 0,C 180,E1 -10917.772,E2 -10917.772} C_VEL
LIN {X 0,Y 556.197,Z 588.137,A -85,B 0,C 180,E1 -10920.248,E2 -10920.248} C_VEL
LIN {X 0,Y 556.18,Z 588.137,A -85,B 0,C 180,E1 -10922.788,E2 -10922.788} C_VEL
LIN {X 0,Y 556.246,Z 588.13,A -85,B 0,C 180,E1 -10925.398,E2 -10925.398} C_VEL
LIN {X 0,Y 556.204,Z 588.128,A -85,B 0,C 180,E1 -10928.103,E2 -10928.103} C_VEL
LIN {X 0,Y 556.196,Z 588.131,A -85,B 0,C 180,E1 -10930.921,E2 -10930.921} C_VEL
LIN {X 0,Y 556.215,Z 588.132,A -85,B 0,C 180,E1 -10933.838,E2 -10933.838} C_VEL
LIN {X 0,Y 556.216,Z 588.131,A -85,B 0,C 180,E1 -10936.162,E2 -10936.162} C_VEL
LIN {X 0,Y 556.235,Z 588.132,A -85,B 0,C 180,E1 -10939.094,E2 -10939.094} C_VEL
LIN {X 0,Y 556.206,Z 588.132,A -85,B 0,C 180,E1 -10941.898,E2 -10941.898} C_VEL
LIN {X 0,Y 556.27,Z 588.126,A -85,B 0,C 180,E1 -10944.604,E2 -10944.604} C_VEL
LIN {X 0,Y 556.206,Z 588.132,A -85,B 0,C 180,E1 -10947.538,E2 -10947.538} C_VEL
LIN {X 0,Y 556.238,Z 588.128,A -85,B 0,C 180,E1 -10950.33,E2 -10950.33} C_VEL
LIN {X 0,Y 556.223,Z 588.134,A -85,B 0,C 180,E1 -10953.042,E2 -10953.042} C_VEL
LIN {X 0,Y 556.229,Z 588.13,A -85,B 0,C 180,E1 -10955.445,E2 -10955.445} C_VEL
LIN {X 0,Y 556.243,Z 588.131,A -85,B 0,C 180,E1 -10957.804,E2 -10957.804} C_VEL
LIN {X 0,Y 556.249,Z 588.135,A -85,B 0,C 180,E1 -10960.889,E2 -10960.889} C_VEL
LIN {X 0,Y 556.234,Z 588.133,A -85,B 0,C 180,E1 -10963.916,E2 -10963.916} C_VEL
LIN {X 0,Y 556.326,Z 588.122,A -85,B 0,C 180,E1 -10966.159,E2 -10966.159} C_VEL
LIN {X 0,Y 556.314,Z 588.254,A -85,B 0,C 180,E1 -10968.332,E2 -10968.332} C_VEL
LIN {X 0,Y 557.928,Z 597.081,A -85,B 0,C 180,E1 -10970.242,E2 -10970.242} C_VEL
LIN {X 0,Y 558.045,Z 602.459,A -85,B 0,C 180,E1 -10971.337,E2 -10971.337} C_VEL
LIN {X 0,Y 557.368,Z 615.368,A -85,B 0,C 180,E1 -10973.868,E2 -10973.868} C_VEL
LIN {X 0,Y 556.753,Z 624.276,A -85,B 0,C 180,E1 -10975.58,E2 -10975.58} C_VEL
LIN {X 0,Y 559.805,Z 641.381,A -85,B 0,C 180,E1 -10975.953,E2 -10975.953} C_VEL
LIN {X 0,Y 558.675,Z 710.829,A -85,B 0,C 180,E1 -10976.99,E2 -10976.99} C_VEL
LIN {X 0,Y 558.354,Z 732.761,A -85,B 0,C 180,E1 -10977.348,E2 -10977.348} C_VEL
LIN {X 0,Y 558.066,Z 746.158,A -85,B 0,C 180,E1 -10977.707,E2 -10977.707} C_VEL
LIN {X 0,Y 557.77,Z 758.562,A -85,B 0,C 180,E1 -10978.201,E2 -10978.201} C_VEL
LIN {X 0,Y 557.496,Z 769.007,A -85,B 0,C 180,E1 -10978.74,E2 -10978.74} C_VEL
LIN {X 0,Y 557.17,Z 778.86,A -85,B 0,C 180,E1 -10979.37,E2 -10979.37} C_VEL
LIN {X 0,Y 556.715,Z 788.174,A -85,B 0,C 180,E1 -10980.09,E2 -10980.09} C_VEL
LIN {X 0,Y 556.298,Z 796.873,A -85,B 0,C 180,E1 -10980.902,E2 -10980.902} C_VEL
LIN {X 0,Y 555.894,Z 803.483,A -85,B 0,C 180,E1 -10981.624,E2 -10981.624} C_VEL
LIN {X 0,Y 555.637,Z 810.393,A -85,B 0,C 180,E1 -10982.529,E2 -10982.529} C_VEL
LIN {X 0,Y 555.28,Z 816.203,A -85,B 0,C 180,E1 -10983.435,E2 -10983.435} C_VEL
LIN {X 0,Y 555.165,Z 822.251,A -85,B 0,C 180,E1 -10984.631,E2 -10984.631} C_VEL
LIN {X 0,Y 555.081,Z 825.6,A -85,B 0,C 180,E1 -10985.43,E2 -10985.43} C_VEL
LIN {X 0,Y 554.948,Z 829.104,A -85,B 0,C 180,E1 -10986.522,E2 -10986.522} C_VEL
LIN {X 0,Y 554.75,Z 832.105,A -85,B 0,C 180,E1 -10987.983,E2 -10987.983} C_VEL
LIN {X 0,Y 554.792,Z 833.073,A -85,B 0,C 180,E1 -10988.714,E2 -10988.714} C_VEL
LIN {X 0,Y 554.788,Z 833.532,A -85,B 0,C 180,E1 -10990.181,E2 -10990.181} C_VEL
LIN {X 0,Y 554.784,Z 833.179,A -85,B 0,C 180,E1 -10990.916,E2 -10990.916} C_VEL
LIN {X 0,Y 554.769,Z 831.109,A -85,B 0,C 180,E1 -10992.394,E2 -10992.394} C_VEL
LIN {X 0,Y 554.924,Z 828.043,A -85,B 0,C 180,E1 -10993.609,E2 -10993.609} C_VEL
LIN {X 0,Y 554.992,Z 824.546,A -85,B 0,C 180,E1 -10994.62,E2 -10994.62} C_VEL
LIN {X 0,Y 555.18,Z 819.476,A -85,B 0,C 180,E1 -10995.739,E2 -10995.739} C_VEL
LIN {X 0,Y 555.3,Z 814.396,A -85,B 0,C 180,E1 -10996.65,E2 -10996.65} C_VEL
LIN {X 0,Y 555.524,Z 807.838,A -85,B 0,C 180,E1 -10997.614,E2 -10997.614} C_VEL
LIN {X 0,Y 555.874,Z 800.079,A -85,B 0,C 180,E1 -10998.552,E2 -10998.552} C_VEL
LIN {X 0,Y 556.202,Z 791.741,A -85,B 0,C 180,E1 -10999.389,E2 -10999.389} C_VEL
LIN {X 0,Y 556.517,Z 782.565,A -85,B 0,C 180,E1 -11000.154,E2 -11000.154} C_VEL
LIN {X 0,Y 556.891,Z 772.977,A -85,B 0,C 180,E1 -11000.813,E2 -11000.813} C_VEL
LIN {X 0,Y 557.193,Z 764.841,A -85,B 0,C 180,E1 -11001.283,E2 -11001.283} C_VEL
LIN {X 0,Y 557.494,Z 753.68,A -85,B 0,C 180,E1 -11001.799,E2 -11001.799} C_VEL
LIN {X 0,Y 557.668,Z 742.817,A -85,B 0,C 180,E1 -11002.184,E2 -11002.184} C_VEL
LIN {X 0,Y 557.921,Z 731.724,A -85,B 0,C 180,E1 -11002.465,E2 -11002.465} C_VEL
LIN {X 0,Y 558.24,Z 712.431,A -85,B 0,C 180,E1 -11002.768,E2 -11002.768} C_VEL
LIN {X 0,Y 558.938,Z 639.965,A -85,B 0,C 180,E1 -11003.82,E2 -11003.82} C_VEL
LIN {X 0,Y 556.387,Z 623.096,A -85,B 0,C 180,E1 -11004.145,E2 -11004.145} C_VEL
LIN {X 0,Y 557.04,Z 607.06,A -85,B 0,C 180,E1 -11007.117,E2 -11007.117} C_VEL
LIN {X 0,Y 557.375,Z 595.199,A -85,B 0,C 180,E1 -11009.347,E2 -11009.347} C_VEL
LIN {X 0,Y 556.319,Z 588.121,A -85,B 0,C 180,E1 -11010.763,E2 -11010.763} C_VEL
LIN {X 0,Y 556.224,Z 588.133,A -85,B 0,C 180,E1 -11013.785,E2 -11013.785} C_VEL
LIN {X 0,Y 556.256,Z 588.127,A -85,B 0,C 180,E1 -11016.303,E2 -11016.303} C_VEL
LIN {X 0,Y 556.192,Z 588.13,A -85,B 0,C 180,E1 -11019.026,E2 -11019.026} C_VEL
LIN {X 0,Y 556.206,Z 588.137,A -85,B 0,C 180,E1 -11021.869,E2 -11021.869} C_VEL
LIN {X 0,Y 556.248,Z 588.124,A -85,B 0,C 180,E1 -11024.843,E2 -11024.843} C_VEL
LIN {X 0,Y 556.211,Z 588.138,A -85,B 0,C 180,E1 -11027.986,E2 -11027.986} C_VEL
LIN {X 0,Y 556.231,Z 588.132,A -85,B 0,C 180,E1 -11030.188,E2 -11030.188} C_VEL
LIN {X 0,Y 556.214,Z 588.128,A -85,B 0,C 180,E1 -11032.809,E2 -11032.809} C_VEL
LIN {X 0,Y 556.239,Z 588.127,A -85,B 0,C 180,E1 -11035.482,E2 -11035.482} C_VEL
LIN {X 0,Y 556.214,Z 588.136,A -85,B 0,C 180,E1 -11038.068,E2 -11038.068} C_VEL
LIN {X 0,Y 556.234,Z 588.126,A -85,B 0,C 180,E1 -11040.586,E2 -11040.586} C_VEL
LIN {X 0,Y 556.22,Z 588.129,A -85,B 0,C 180,E1 -11043.392,E2 -11043.392} C_VEL
LIN {X 0,Y 556.227,Z 588.131,A -85,B 0,C 180,E1 -11046.236,E2 -11046.236} C_VEL
LIN {X 0,Y 556.253,Z 588.123,A -85,B 0,C 180,E1 -11048.719,E2 -11048.719} C_VEL
LIN {X 0,Y 556.244,Z 588.129,A -85,B 0,C 180,E1 -11051.65,E2 -11051.65} C_VEL
LIN {X 0,Y 556.279,Z 588.121,A -85,B 0,C 180,E1 -11053.35,E2 -11053.35} C_VEL
LIN {X 0,Y 555.586,Z 588.216,A -85,B 0,C 180,E1 -11053.954,E2 -11053.954} C_VEL
LIN {X 0,Y 552.741,Z 588.569,A -85,B 0,C 180,E1 -11054.936,E2 -11054.936} C_VEL
LIN {X 0,Y 550.352,Z 588.865,A -85,B 0,C 180,E1 -11055.726,E2 -11055.726} C_VEL
LIN {X 0,Y 549.326,Z 588.99,A -85,B 0,C 180,E1 -11056.336,E2 -11056.336} C_VEL
LIN {X 0,Y 549.241,Z 588.998,A -85,B 0,C 180,E1 -11056.542,E2 -11056.542} C_VEL
LIN {X 0,Y 549.291,Z 588.996,A -85,B 0,C 180,E1 -11059.716,E2 -11059.716} C_VEL
LIN {X 0,Y 549.331,Z 588.986,A -85,B 0,C 180,E1 -11062.674,E2 -11062.674} C_VEL
LIN {X 0,Y 549.399,Z 588.977,A -85,B 0,C 180,E1 -11064.88,E2 -11064.88} C_VEL
LIN {X 0,Y 549.178,Z 589.004,A -85,B 0,C 180,E1 -11067.075,E2 -11067.075} C_VEL
LIN {X 0,Y 549.544,Z 588.968,A -85,B 0,C 180,E1 -11070,E2 -11070} C_VEL
LIN {X 0,Y 549.332,Z 588.99,A -85,B 0,C 180,E1 -11073.655,E2 -11073.655} C_VEL
LIN {X 0,Y 549.375,Z 588.989,A -85,B 0,C 180,E1 -11076.024,E2 -11076.024} C_VEL
LIN {X 0,Y 549.274,Z 588.992,A -85,B 0,C 180,E1 -11078.802,E2 -11078.802} C_VEL
LIN {X 0,Y 549.299,Z 588.989,A -85,B 0,C 180,E1 -11081.027,E2 -11081.027} C_VEL
LIN {X 0,Y 549.287,Z 588.995,A -85,B 0,C 180,E1 -11084.273,E2 -11084.273} C_VEL
LIN {X 0,Y 549.236,Z 588.997,A -85,B 0,C 180,E1 -11087.057,E2 -11087.057} C_VEL
LIN {X 0,Y 549.196,Z 589.009,A -85,B 0,C 180,E1 -11090.142,E2 -11090.142} C_VEL
LIN {X 0,Y 549.198,Z 589.004,A -85,B 0,C 180,E1 -11092.496,E2 -11092.496} C_VEL
LIN {X 0,Y 549.168,Z 589.006,A -85,B 0,C 180,E1 -11095.1,E2 -11095.1} C_VEL
LIN {X 0,Y 549.203,Z 589.008,A -85,B 0,C 180,E1 -11098.157,E2 -11098.157} C_VEL
LIN {X 0,Y 549.202,Z 589.002,A -85,B 0,C 180,E1 -11100.674,E2 -11100.674} C_VEL
LIN {X 0,Y 549.2,Z 589.011,A -85,B 0,C 180,E1 -11104.004,E2 -11104.004} C_VEL
LIN {X 0,Y 549.218,Z 588.999,A -85,B 0,C 180,E1 -11106.828,E2 -11106.828} C_VEL
LIN {X 0,Y 549.198,Z 589.01,A -85,B 0,C 180,E1 -11110.073,E2 -11110.073} C_VEL
LIN {X 0,Y 549.185,Z 589.005,A -85,B 0,C 180,E1 -11113.366,E2 -11113.366} C_VEL
LIN {X 0,Y 549.193,Z 589.006,A -85,B 0,C 180,E1 -11115.58,E2 -11115.58} C_VEL
LIN {X 0,Y 549.172,Z 589.005,A -85,B 0,C 180,E1 -11118.809,E2 -11118.809} C_VEL
LIN {X 0,Y 549.17,Z 589.006,A -85,B 0,C 180,E1 -11121.32,E2 -11121.32} C_VEL
LIN {X 0,Y 549.232,Z 589.005,A -85,B 0,C 180,E1 -11124.081,E2 -11124.081} C_VEL
LIN {X 0,Y 549.163,Z 589.007,A -85,B 0,C 180,E1 -11126.739,E2 -11126.739} C_VEL
LIN {X 0,Y 549.184,Z 589.005,A -85,B 0,C 180,E1 -11129.325,E2 -11129.325} C_VEL
LIN {X 0,Y 549.204,Z 589.009,A -85,B 0,C 180,E1 -11131.843,E2 -11131.843} C_VEL
LIN {X 0,Y 549.171,Z 589.005,A -85,B 0,C 180,E1 -11134.901,E2 -11134.901} C_VEL
LIN {X 0,Y 549.199,Z 589.004,A -85,B 0,C 180,E1 -11137.504,E2 -11137.504} C_VEL
LIN {X 0,Y 549.192,Z 589.01,A -85,B 0,C 180,E1 -11139.858,E2 -11139.858} C_VEL
LIN {X 0,Y 549.205,Z 589.001,A -85,B 0,C 180,E1 -11143.045,E2 -11143.045} C_VEL
LIN {X 0,Y 549.282,Z 589.001,A -85,B 0,C 180,E1 -11145.979,E2 -11145.979} C_VEL
LIN {X 0,Y 549.324,Z 588.986,A -85,B 0,C 180,E1 -11149.061,E2 -11149.061} C_VEL
LIN {X 0,Y 549.304,Z 588.998,A -85,B 0,C 180,E1 -11151.937,E2 -11151.937} C_VEL
LIN {X 0,Y 549.368,Z 588.987,A -85,B 0,C 180,E1 -11154.146,E2 -11154.146} C_VEL
LIN {X 0,Y 549.326,Z 588.989,A -85,B 0,C 180,E1 -11156.345,E2 -11156.345} C_VEL
LIN {X 0,Y 549.547,Z 588.967,A -85,B 0,C 180,E1 -11160,E2 -11160} C_VEL
LIN {X 0,Y 549.325,Z 588.991,A -85,B 0,C 180,E1 -11163.656,E2 -11163.656} C_VEL
LIN {X 0,Y 549.399,Z 588.985,A -85,B 0,C 180,E1 -11166.043,E2 -11166.043} C_VEL
LIN {X 0,Y 549.281,Z 588.992,A -85,B 0,C 180,E1 -11168.802,E2 -11168.802} C_VEL
LIN {X 0,Y 549.303,Z 588.989,A -85,B 0,C 180,E1 -11171.027,E2 -11171.027} C_VEL
LIN {X 0,Y 549.276,Z 588.997,A -85,B 0,C 180,E1 -11174.266,E2 -11174.266} C_VEL
LIN {X 0,Y 549.185,Z 589.003,A -85,B 0,C 180,E1 -11177.059,E2 -11177.059} C_VEL
LIN {X 0,Y 549.171,Z 589.012,A -85,B 0,C 180,E1 -11180.144,E2 -11180.144} C_VEL
LIN {X 0,Y 549.189,Z 589.005,A -85,B 0,C 180,E1 -11182.496,E2 -11182.496} C_VEL
LIN {X 0,Y 549.171,Z 589.005,A -85,B 0,C 180,E1 -11185.099,E2 -11185.099} C_VEL
LIN {X 0,Y 549.203,Z 589.007,A -85,B 0,C 180,E1 -11188.157,E2 -11188.157} C_VEL
LIN {X 0,Y 549.161,Z 589.007,A -85,B 0,C 180,E1 -11190.677,E2 -11190.677} C_VEL
LIN {X 0,Y 549.124,Z 589.012,A -85,B 0,C 180,E1 -11193.264,E2 -11193.264} C_VEL
LIN {X 0,Y 549.174,Z 589.014,A -85,B 0,C 180,E1 -11195.924,E2 -11195.924} C_VEL
LIN {X 0,Y 549.125,Z 589.011,A -85,B 0,C 180,E1 -11198.914,E2 -11198.914} C_VEL
LIN {X 0,Y 549.149,Z 589.011,A -85,B 0,C 180,E1 -11201.549,E2 -11201.549} C_VEL
LIN {X 0,Y 549.199,Z 589.003,A -85,B 0,C 180,E1 -11204.545,E2 -11204.545} C_VEL
LIN {X 0,Y 549.149,Z 589.01,A -85,B 0,C 180,E1 -11207.467,E2 -11207.467} C_VEL
LIN {X 0,Y 549.132,Z 589.013,A -85,B 0,C 180,E1 -11210.374,E2 -11210.374} C_VEL
LIN {X 0,Y 549.157,Z 589.009,A -85,B 0,C 180,E1 -11213.471,E2 -11213.471} C_VEL
LIN {X 0,Y 549.144,Z 589.017,A -85,B 0,C 180,E1 -11216.005,E2 -11216.005} C_VEL
LIN {X 0,Y 549.156,Z 589.008,A -85,B 0,C 180,E1 -11218.713,E2 -11218.713} C_VEL
LIN {X 0,Y 549.175,Z 589.009,A -85,B 0,C 180,E1 -11221.649,E2 -11221.649} C_VEL
LIN {X 0,Y 549.132,Z 589.019,A -85,B 0,C 180,E1 -11224.298,E2 -11224.298} C_VEL
LIN {X 0,Y 549.188,Z 589.036,A -85,B 0,C 180,E1 -11226.048,E2 -11226.048} C_VEL
LIN {X 0,Y 551.24,Z 600.431,A -85,B 0,C 180,E1 -11228.062,E2 -11228.062} C_VEL
LIN {X 0,Y 550.93,Z 610.42,A -85,B 0,C 180,E1 -11229.73,E2 -11229.73} C_VEL
LIN {X 0,Y 549.973,Z 628.96,A -85,B 0,C 180,E1 -11232.784,E2 -11232.784} C_VEL
LIN {X 0,Y 549.259,Z 646.984,A -85,B 0,C 180,E1 -11235.723,E2 -11235.723} C_VEL
LIN {X 0,Y 551.883,Z 669.615,A -85,B 0,C 180,E1 -11236.14,E2 -11236.14} C_VEL
LIN {X 0,Y 550.971,Z 754.103,A -85,B 0,C 180,E1 -11237.402,E2 -11237.402} C_VEL
LIN {X 0,Y 550.737,Z 763.98,A -85,B 0,C 180,E1 -11237.63,E2 -11237.63} C_VEL
LIN {X 0,Y 550.471,Z 774.601,A -85,B 0,C 180,E1 -11237.974,E2 -11237.974} C_VEL
LIN {X 0,Y 550.158,Z 784.729,A -85,B 0,C 180,E1 -11238.403,E2 -11238.403} C_VEL
LIN {X 0,Y 549.951,Z 793.584,A -85,B 0,C 180,E1 -11238.868,E2 -11238.868} C_VEL
LIN {X 0,Y 549.512,Z 803.903,A -85,B 0,C 180,E1 -11239.535,E2 -11239.535} C_VEL
LIN {X 0,Y 549.204,Z 812.193,A -85,B 0,C 180,E1 -11240.178,E2 -11240.178} C_VEL
LIN {X 0,Y 548.782,Z 821.046,A -85,B 0,C 180,E1 -11241.005,E2 -11241.005} C_VEL
LIN {X 0,Y 548.504,Z 827.753,A -85,B 0,C 180,E1 -11241.74,E2 -11241.74} C_VEL
LIN {X 0,Y 548.239,Z 834.777,A -85,B 0,C 180,E1 -11242.66,E2 -11242.66} C_VEL
LIN {X 0,Y 548.036,Z 841.622,A -85,B 0,C 180,E1 -11243.763,E2 -11243.763} C_VEL
LIN {X 0,Y 547.949,Z 845.505,A -85,B 0,C 180,E1 -11244.499,E2 -11244.499} C_VEL
LIN {X 0,Y 547.811,Z 850.851,A -85,B 0,C 180,E1 -11245.807,E2 -11245.807} C_VEL
LIN {X 0,Y 547.777,Z 853.69,A -85,B 0,C 180,E1 -11246.701,E2 -11246.701} C_VEL
LIN {X 0,Y 547.773,Z 856.181,A -85,B 0,C 180,E1 -11247.802,E2 -11247.802} C_VEL
LIN {X 0,Y 547.729,Z 857.928,A -85,B 0,C 180,E1 -11249.267,E2 -11249.267} C_VEL
LIN {X 0,Y 547.718,Z 858.241,A -85,B 0,C 180,E1 -11250,E2 -11250} C_VEL
LIN {X 0,Y 547.722,Z 857.543,A -85,B 0,C 180,E1 -11251.466,E2 -11251.466} C_VEL
LIN {X 0,Y 547.773,Z 856.532,A -85,B 0,C 180,E1 -11252.199,E2 -11252.199} C_VEL
LIN {X 0,Y 547.798,Z 853.344,A -85,B 0,C 180,E1 -11253.666,E2 -11253.666} C_VEL
LIN {X 0,Y 547.855,Z 849.706,A -85,B 0,C 180,E1 -11254.767,E2 -11254.767} C_VEL
LIN {X 0,Y 548.017,Z 844.93,A -85,B 0,C 180,E1 -11255.869,E2 -11255.869} C_VEL
LIN {X 0,Y 548.228,Z 838.857,A -85,B 0,C 180,E1 -11256.972,E2 -11256.972} C_VEL
LIN {X 0,Y 548.478,Z 832.712,A -85,B 0,C 180,E1 -11257.891,E2 -11257.891} C_VEL
LIN {X 0,Y 548.76,Z 825.318,A -85,B 0,C 180,E1 -11258.811,E2 -11258.811} C_VEL
LIN {X 0,Y 549.305,Z 816.356,A -85,B 0,C 180,E1 -11259.727,E2 -11259.727} C_VEL
LIN {X 0,Y 549.722,Z 807.779,A -85,B 0,C 180,E1 -11260.461,E2 -11260.461} C_VEL
LIN {X 0,Y 550.134,Z 798.562,A -85,B 0,C 180,E1 -11261.12,E2 -11261.12} C_VEL
LIN {X 0,Y 550.544,Z 787.781,A -85,B 0,C 180,E1 -11261.746,E2 -11261.746} C_VEL
LIN {X 0,Y 550.891,Z 777.974,A -85,B 0,C 180,E1 -11262.204,E2 -11262.204} C_VEL
LIN {X 0,Y 551.211,Z 767.256,A -85,B 0,C 180,E1 -11262.592,E2 -11262.592} C_VEL
LIN {X 0,Y 551.558,Z 755.881,A -85,B 0,C 180,E1 -11262.887,E2 -11262.887} C_VEL
LIN {X 0,Y 551.906,Z 734.849,A -85,B 0,C 180,E1 -11263.229,E2 -11263.229} C_VEL
LIN {X 0,Y 552.729,Z 668.167,A -85,B 0,C 180,E1 -11264.253,E2 -11264.253} C_VEL
LIN {X 0,Y 550.193,Z 649.852,A -85,B 0,C 180,E1 -11264.637,E2 -11264.637} C_VEL
LIN {X 0,Y 549.576,Z 646.06,A -85,B 0,C 180,E1 -11264.739,E2 -11264.739} C_VEL
LIN {X 0,Y 550.519,Z 626.755,A -85,B 0,C 180,E1 -11267.971,E2 -11267.971} C_VEL
LIN {X 0,Y 551.656,Z 608.999,A -85,B 0,C 180,E1 -11271.02,E2 -11271.02} C_VEL
LIN {X 0,Y 551.844,Z 602.935,A -85,B 0,C 180,E1 -11272.093,E2 -11272.093} C_VEL
LIN {X 0,Y 549.514,Z 590.654,A -85,B 0,C 180,E1 -11274.473,E2 -11274.473} C_VEL
LIN {X 0,Y 549.194,Z 589.01,A -85,B 0,C 180,E1 -11274.84,E2 -11274.84} C_VEL
LIN {X 0,Y 549.164,Z 589.017,A -85,B 0,C 180,E1 -11277.334,E2 -11277.334} C_VEL
